//With this function its possible to control a heating pump with the plc
//When the heating pump is switching maualy, then the target power from the ems function is without functionality
//On the max power inputs can be add the power limits. The pump can by step switched by 2 steps
//The percent number from each step is added to the output target power
//< Constants.byTargetOffPowerOnOffDevices Target power from the ems dissable the heating pump after the delay in the surplus mode in Step 4
//When the HP is not step switched, the input target power is set linear to the output target power.
//When the target power from the ems <= 0 and after delay then the heating pump is dissabled in the surplus mode in step 4
//On the emergency power mode and when the soc from the battery <= dissableSOC then the target output power from the heating pump is 0
//Otherwise the heating pump runs in normal mode and the output boutputHB is then always true 
//If in the setups from the heating pump the OffOn Emergency mode is true then the Heating pump is dissabled in the emergency power mode
//When the time function is enabled, then the heating pump run in this time with the % value from max power [1] from the setup when its step switched.
//If there is no step switching and time mode is active, the power input is set linearly to the output. The % value with which the pump should then run over the time can be set at the setups
//This function has also a external look input. If this input is set then the heating pump is dissabled
//This function has also a step to activate the heating pump by a external command. Here the pump switch on with delay and check before the power on the grid

(*---------------------------------------------------------------Limits-------------------------------------------------------------------------------*)

dwBatterySOC := LIMIT(0,dwBatterySOC,100);
	stSetupHP.byManualyTargetPower := LIMIT(0,stSetupHP.byManualyTargetPower,100);
		rBoilerTempHeatingSys := LIMIT(-30,rBoilerTempHeatingSys,120);
			rBoilerTempServiceWater := LIMIT(-30,rBoilerTempServiceWater,120);
				rFlowTemp := LIMIT(-30,rFlowTemp,120);
					rReturnTemp := LIMIT(-30,rReturnTemp,120);
						rFlowTempEnergySource := LIMIT(-30,rFlowTempEnergySource,120); 
							rReturnTempEnergySource := LIMIT(-30,rReturnTempEnergySource,120); 
								stSetupHP.byTimeEnabledTargetPower := LIMIT(0,stSetupHP.byTimeEnabledTargetPower,100);
									stSetupHP.byHourOn := LIMIT(0,stSetupHP.byHourOn,23);
										stSetupHP.byHourOff := LIMIT(0,stSetupHP.byHourOff,23);
											stSetupHP.byMinutesOn := LIMIT(0,stSetupHP.byMinutesOn,59);
												stSetupHP.byMinutesOff := LIMIT(0,stSetupHP.byMinutesOff,59);
													IF IsFinite(F_LREAL(lrCounterThermalEnergy_Water)) THEN lrCounterThermalEnergy_Water := LIMIT(0,lrCounterThermalEnergy_Water,999999999999999); END_IF
														IF IsFinite(F_LREAL(lrCounterThermalEnergy_Heating)) THEN lrCounterThermalEnergy_Heating := LIMIT(0,lrCounterThermalEnergy_Heating,999999999999999); END_IF
															diNumberOfHP := LIMIT(0,diNumberOfHP,Constants_Energy.diMaxNumberOfHeatingPumps);
																tOnDelayExternalOn := LIMIT(T#1M,tOnDelayExternalOn,T#10M);	
																	tOffDelayExternalOn := LIMIT(T#15M,tOffDelayExternalOn,T#2H);
																		tMinOnTime := LIMIT(T#15M,tMinOnTime,T#2H);	

IF IsFinite(F_LREAL(lrTotalCounterEnergy_Consumption)) THEN lrTotalCounterEnergy_Consumption := LIMIT(0,lrTotalCounterEnergy_Consumption,999999999999999); END_IF
	IF IsFinite(F_LREAL(lrTotalCounterEnergy_Production)) THEN lrTotalCounterEnergy_Production := LIMIT(0,lrTotalCounterEnergy_Production,999999999999999); END_IF
		IF IsFinite(F_LREAL(lrCounterEnergyT1_Consumption)) THEN lrCounterEnergyT1_Consumption := LIMIT(0,lrCounterEnergyT1_Consumption,999999999999999); END_IF
			IF IsFinite(F_LREAL(lrCounterEnergyT2_Consumption)) THEN lrCounterEnergyT2_Consumption := LIMIT(0,lrCounterEnergyT2_Consumption,999999999999999); END_IF
				IF IsFinite(F_LREAL(lrCounterEnergyT1_Production)) THEN lrCounterEnergyT1_Production := LIMIT(0,lrCounterEnergyT1_Production,999999999999999); END_IF
					IF IsFinite(F_LREAL(lrCounterEnergyT2_Production)) THEN lrCounterEnergyT2_Production := LIMIT(0,lrCounterEnergyT2_Production,999999999999999); END_IF
						lrElPowerHP := LIMIT(-999999999999999,lrElPowerHP,999999999999999);	
							lrSizeGridConnection := LIMIT(-999999999999999,lrSizeGridConnection,999999999999999);	
								lrGridPower := LIMIT(-999999999999999,lrGridPower,999999999999999);														
														
IF bIsStepSwitched AND stSetupHP.rMaxPower1 <= 0 AND stSetupHP.rMaxPower2 > 0 THEN stSetupHP.rMaxPower1 := stSetupHP.rMaxPower2; END_IF												
												
FOR byLPMaxPower := 1 TO 2 BY 1 DO
	arrTargetPower[byLPMaxPower] := LIMIT(0,arrTargetPower[byLPMaxPower],100);
END_FOR

stSetupHP.rMaxPower1 := LIMIT(0,stSetupHP.rMaxPower1,500);
		stSetupHP.rMaxPower2 := LIMIT(0,stSetupHP.rMaxPower2,500);

//Copy the max input power in the internal array to calculate the steps
arrMaxPower[1] := stSetupHP.rMaxPower1;
	arrMaxPower[2] := stSetupHP.rMaxPower2;
	
IF stSetupHP.byDisableSOC > stSetupHP.byEnableSOC THEN stSetupHP.byEnableSOC := stSetupHP.byDisableSOC + 1; END_IF

stSetupHP.byDisableSOC := LIMIT(0,stSetupHP.byDisableSOC,100);
	stSetupHP.byEnableSOC := LIMIT(1,stSetupHP.byEnableSOC,100);
	
(*---------------------------------------------------------------------------Enable----------------------------------------------------------------------------------*)

stDataHPOut.bEnabled := bEnable;

(*-----------------------------------------------------------------------------Count the steps when the pump is step switched----------------------------------------------------------------------------*)

stDataHPOut.byNumberOfSteps := 0;
	FOR byLPNumberOfSteps := 1 TO 2 BY 1 DO
		IF arrMaxPower[byLPNumberOfSteps] > 0 THEN stDataHPOut.byNumberOfSteps := stDataHPOut.byNumberOfSteps + 1; END_IF
	END_FOR

(*-----------------------------------------------------------------------------Max power for the output----------------------------------------------------------------------------*)	
	
FOR byLPMaxPowerLimit := 1 TO 2 BY 1 DO
	stDataHPOut.arrMaxPower[byLPMaxPowerLimit] := DINT_TO_REAL(REAL_TO_DINT(arrMaxPower[byLPMaxPowerLimit] * 100)) / 100;
END_FOR		
	
(*-----------------------------------------------------------------------------Errors and Warning----------------------------------------------------------------------------*)

FPReset(CLK:= stSetupHP.bReset AND (stDataHPOut.byErrorWarning <> 0), Q=> ); 
	timResetOut(IN:= FPReset.Q AND NOT timResetOut.Q, PT:= T#2S, Q=> stDataHPOut.bSReset, ET=> );
		FPResetIntern(CLK:= bReset, Q=> );	
			IF FPResetIntern.Q THEN stDataHPOut.byErrorWarning := 0; END_IF	 	

IF bWarning AND stDataHPOut.byErrorWarning <> 2 THEN stDataHPOut.byErrorWarning := 1; END_IF
	IF bError THEN stDataHPOut.byErrorWarning := 2; END_IF

//Messages and Error Codes
IF uiState = 3 THEN stDataHPOut.eMessage := E_Message_HP.eExternalOnCommandIsActive;	
ELSIF bExternalLock THEN stDataHPOut.eMessage := E_Message_HP.eExternalLockActive;
ELSIF stDataHPOut.byErrorWarning = 1 AND iWarningCode = 0 THEN stDataHPOut.eMessage := E_Message_HP.eNoConnectionToBackend;
ELSIF stDataHPOut.byErrorWarning = 2 AND iErrorCode = 0 THEN stDataHPOut.eMessage := E_Message_HP.eHPError;
ELSIF stDataHPOut.byErrorWarning = 2 AND iErrorCode = 1 THEN stDataHPOut.eMessage := E_Message_HP.eTooMuchHP;
ELSIF stDataHPOut.byErrorWarning = 2 AND iErrorCode = 2 THEN stDataHPOut.eMessage := E_Message_HP.eWindowsSystemTimeError;
ELSIF stDataHPOut.byErrorWarning = 2 AND iErrorCode = 3 THEN stDataHPOut.eMessage := E_Message_HP.eConnectionError;
ELSE stDataHPOut.eMessage := E_Message_HP.eNoMessage; 
END_IF	
	
(*----------------------------------------------------------------------------Logic------------------------------------------------------------------------------------*)

//Timer for SOC dissabling
timSOCOff(IN:= dwBatterySOC <= stSetupHP.byDisableSOC, PT:= T#30S, Q=> , ET=> );

//Calcualte the % value from each step when the pump is step switched
rSumOfSteps := 0;
	FOR byLPCalcStepPower := 1 TO 2 BY 1 DO
		rSumOfSteps := rSumOfSteps + stDataHPOut.arrMaxPower[byLPCalcStepPower];
			arrPercentValuesSteps[byLPCalcStepPower] := 0;	
	END_FOR
IF stDataHPOut.byNumberOfSteps > 0 AND stDataHPOut.byNumberOfSteps <= 2 AND rSumOfSteps > 0 THEN
	FOR byLPCalcPercentPowerSteps := 1 TO stDataHPOut.byNumberOfSteps BY 1 DO
		arrPercentValuesSteps[byLPCalcPercentPowerSteps] := (stDataHPOut.arrMaxPower[byLPCalcPercentPowerSteps] * 100) / rSumOfSteps;
	END_FOR 
END_IF

arrPercentValuesSteps[1] := DINT_TO_REAL(REAL_TO_DINT(arrPercentValuesSteps[1] * 100)) / 100; 
	arrPercentValuesSteps[2] := DINT_TO_REAL(REAL_TO_DINT(arrPercentValuesSteps[2] * 100)) / 100; 

//Enable the pump about the time function
FPTimeEn(CLK:= stSystemTime.wHour >= stSetupHP.byHourOn AND stSystemTime.wMinute >= stSetupHP.byMinutesOn AND stSetupHP.bTimeEnabled, Q=> );
	FPTimeDis(CLK:= stSystemTime.wHour >= stSetupHP.byHourOff AND stSystemTime.wMinute >= stSetupHP.byMinutesOff AND stSetupHP.bTimeEnabled, Q=> );

IF FPTimeEn.Q THEN bEnableTimeFunction := TRUE; END_IF
	IF FPTimeDis.Q THEN bEnableTimeFunction := FALSE; END_IF	
	
IF NOT stSetupHP.bTimeEnabled THEN bEnableTimeFunction := FALSE; END_IF

//Activate the different operation modes

FPExternalOnCommand(CLK:= bExternalOnCommand, Q=> );

IF bEnable AND NOT bExternalLock AND bEnableTimeFunction AND NOT bIsStepSwitched AND stDataHPOut.byErrorWarning <> 2 THEN uiState := 1; END_IF
IF bEnable AND NOT bExternalLock AND bEnableTimeFunction AND bIsStepSwitched AND stDataHPOut.byErrorWarning <> 2 THEN uiState := 2; END_IF
IF bEnable AND NOT bExternalLock AND NOT bEPOIsActive AND FPExternalOnCommand.Q AND stDataHPOut.byErrorWarning <> 2 THEN uiState := 3; END_IF
IF bEnable AND NOT bExternalLock AND stDataHPOut.byErrorWarning <> 2 AND (arrTargetPower[1] > 0 OR arrTargetPower[2] > 0) THEN uiState := 4; END_IF
IF bEnable AND NOT bExternalLock AND stDataHPOut.byErrorWarning <> 2 AND stSetupHP.bManualyOn THEN uiState := 5; END_IF 

IF NOT bEnable OR stDataHPOut.byErrorWarning = 2 OR bExternalLock THEN uiState := 0; END_IF

//Timer for Min on time in Step 4 in the surplus mode
FPStartMinOnTimer(CLK:= uiState = 4 AND stDataHPOut.rTargetPower > 0 AND bHPIsRunning, Q=> );
	timMinOnInStep4(IN:= FPStartMinOnTimer.Q, PT:= tMinOnTime, Q=> , ET=> );

CASE uiState OF
	
	0: //Init Step and Error
		IF (NOT bEPOIsActive AND bEnable AND NOT bExternalLock AND stDataHPOut.byErrorWarning <> 2) OR 
				(bEPOIsActive AND bEnable AND NOT bExternalLock AND stDataHPOut.byErrorWarning <> 2 AND NOT stSetupHP.bOnEmergPowerOff AND dwBatterySOC >= stSetupHP.byEnableSOC) THEN
					stDataHPOut.bOutput := TRUE;
		END_IF
			IF (bEPOIsActive AND timSOCOff.Q OR NOT bEnable OR bExternalLock OR stDataHPOut.byErrorWarning = 2 OR (bEPOIsActive AND stSetupHP.bOnEmergPowerOff)) THEN
				stDataHPOut.bOutput := FALSE;
					stDataHPOut.rTargetPower := 0;
			END_IF
			
	1: //Enable Heating pump about the time function (linear power)
		//On
		IF (NOT bEPOIsActive AND bEnableTimeFunction AND stSetupHP.byTimeEnabledTargetPower > 0) OR (bEnableTimeFunction AND stSetupHP.byTimeEnabledTargetPower > 0 AND bEPOIsActive AND NOT stSetupHP.bOnEmergPowerOff AND dwBatterySOC >= stSetupHP.byEnableSOC) THEN
			stDataHPOut.bOutput := TRUE; stDataHPOut.rTargetPower := BYTE_TO_REAL(stSetupHP.byTimeEnabledTargetPower);
		END_IF
		//Off		
		IF NOT bEnableTimeFunction OR stSetupHP.byTimeEnabledTargetPower <= 0 OR (bEPOIsActive AND stSetupHP.bOnEmergPowerOff) OR (bEPOIsActive AND (timSOCOff.Q)) THEN 
			stDataHPOut.rTargetPower := 0; 
		END_IF	
			IF stSetupHP.byTimeEnabledTargetPower <= 0 OR (bEPOIsActive AND stSetupHP.bOnEmergPowerOff) OR (bEPOIsActive AND (timSOCOff.Q)) THEN
				stDataHPOut.bOutput := FALSE;
			END_IF	 
		
	2: //Enable Heating pump about the time function (step switched)
		//On
		IF (NOT bEPOIsActive AND bEnableTimeFunction AND arrPercentValuesSteps[1] > 0) OR (bEnableTimeFunction AND arrPercentValuesSteps[1] > 0 AND bEPOIsActive AND NOT stSetupHP.bOnEmergPowerOff AND dwBatterySOC >= stSetupHP.byEnableSOC) THEN
			stDataHPOut.bOutput := TRUE; stDataHPOut.rTargetPower := arrPercentValuesSteps[1];
		END_IF
		//Off
		IF NOT bEnableTimeFunction OR arrPercentValuesSteps[1] <= 0 OR (bEPOIsActive AND stSetupHP.bOnEmergPowerOff) OR (bEPOIsActive AND (timSOCOff.Q)) THEN 
			stDataHPOut.rTargetPower := 0; 
		END_IF	
			IF arrPercentValuesSteps[1] <= 0 OR (bEPOIsActive AND stSetupHP.bOnEmergPowerOff) OR (bEPOIsActive AND (timSOCOff.Q)) THEN
				stDataHPOut.bOutput := FALSE;
			END_IF	 
	 
	3: //Switch on the HP with external on command on max power
		
			CASE iStateIntStep3 OF
				
				0: //Search biggest power from the HP
					//Max Power 1 (1 Step switched or linear/modular)
					IF stSetupHP.rMaxPower1 > 0 AND stSetupHP.rMaxPower2 = 0 THEN
						//Start delay timer when the actual grid power has the capacity for the heating pump max power
						IF (lrGridPower + stSetupHP.rMaxPower1) <= lrSizeGridConnection AND diNumberOfHP > 0 THEN timOnDelayExternalOn.IN := TRUE; ELSE timOnDelayExternalOn.IN := FALSE; END_IF 
					END_IF 
						//Max Power 2 (1 Step switched or linear/modular) 
						IF stSetupHP.rMaxPower2 > 0 AND stSetupHP.rMaxPower1 = 0 THEN 
							//Start delay timer when the actual grid power has the capacity for the heating pump max power
							IF (lrGridPower + stSetupHP.rMaxPower2) <= lrSizeGridConnection AND diNumberOfHP > 0 THEN timOnDelayExternalOn.IN := TRUE; ELSE timOnDelayExternalOn.IN := FALSE; END_IF
						END_IF 
							//Max Power 1 and Max Power 2 (2 Step switched)
							IF stSetupHP.rMaxPower2 > 0 AND stSetupHP.rMaxPower1 > 0 THEN 
								//Start delay timer when the actual grid power has the capacity for the heating pump max power
								IF (lrGridPower + stSetupHP.rMaxPower1 + stSetupHP.rMaxPower2) <= lrSizeGridConnection AND diNumberOfHP > 0 THEN timOnDelayExternalOn.IN := TRUE; ELSE timOnDelayExternalOn.IN := FALSE; END_IF
							END_IF 
								//Next step
								IF timOnDelayExternalOn.Q THEN iStateIntStep3 := 1; timOnDelayExternalOn.IN := FALSE; END_IF
		
				1: //Switch on the Heating pump with max power			
					stDataHPOut.rTargetPower := 100;
						stDataHPOut.bOutput := TRUE;
							stDataHPOut.bExtOnCommandIsActive := TRUE;
								timOffDelayExternalOn.IN := TRUE;
						//Next step
						IF timOffDelayExternalOn.Q THEN iStateIntStep3 := 0; uiState := 0; stDataHPOut.rTargetPower := 0; END_IF 
				
			END_CASE
		
				//Stop this program when the emergency power mode is active
				IF bEPOIsActive THEN uiState := 0; stDataHPOut.rTargetPower := 0; END_IF
					//Stop this programm when we have no power data from the heating pump
					IF stSetupHP.rMaxPower1 >= stSetupHP.rMaxPower2 AND stSetupHP.rMaxPower1 = 0 THEN uiState := 0; stDataHPOut.rTargetPower := 0; END_IF   	
			
	4: //Enable the Heating pump with the target power from the EMS function
		//Power to the heating pump (linear)
		IF NOT bIsStepSwitched AND stDataHPOut.byNumberOfSteps > 0 THEN	
			stDataHPOut.rTargetPower := DINT_TO_REAL(REAL_TO_DINT(arrTargetPower[1] * 100)) / 100;
		END_IF
			//When the min on Time is not passed and the input target power is < 1% then set the output target power to 1%
			IF NOT bIsStepSwitched AND stDataHPOut.byNumberOfSteps > 0 AND arrTargetPower[1] <= 1 AND timMinOnInStep4.Q THEN
				stDataHPOut.rTargetPower := 1;
			END_IF   
		
				//Power to the heating pump (step switched)
				FOR byLPMaxIsReached := 1 TO 2 BY 1 DO
					IF arrTargetPower[byLPMaxIsReached] >= 100 THEN arrMaxIsReached[byLPMaxIsReached] := TRUE; END_IF
						IF arrTargetPower[byLPMaxIsReached] < Constants_Energy.byTargetOffPowerForOnOffDevices THEN arrMaxIsReached[byLPMaxIsReached] := FALSE; END_IF	
				END_FOR
				
				//Off after min on time is passed
				IF NOT timMinOnInStep4.Q AND bIsStepSwitched AND stDataHPOut.byNumberOfSteps > 0 AND NOT arrMaxIsReached[1] AND arrTargetPower[1] < Constants_Energy.byTargetOffPowerForOnOffDevices THEN 
					stDataHPOut.rTargetPower := 0; 
				END_IF
				IF timMinOnInStep4.Q AND bIsStepSwitched AND stDataHPOut.byNumberOfSteps > 0 AND NOT arrMaxIsReached[1] AND arrTargetPower[1] < Constants_Energy.byTargetOffPowerForOnOffDevices THEN 
					stDataHPOut.rTargetPower := arrPercentValuesSteps[1];
				END_IF 
					//Step 1
					IF bIsStepSwitched AND stDataHPOut.byNumberOfSteps > 0 AND arrMaxIsReached[1] AND arrTargetPower[1] >= Constants_Energy.byTargetOffPowerForOnOffDevices THEN 
						stDataHPOut.rTargetPower := arrPercentValuesSteps[1]; 	
					END_IF
						//Step 2
						IF bIsStepSwitched AND stDataHPOut.byNumberOfSteps > 0 AND arrMaxIsReached[1] AND arrMaxIsReached[2] AND arrTargetPower[2] >= Constants_Energy.byTargetOffPowerForOnOffDevices THEN 
							stDataHPOut.rTargetPower := arrPercentValuesSteps[1] + arrPercentValuesSteps[2]; 
						END_IF
						
		IF bIsStepSwitched AND stDataHPOut.rTargetPower > 100 THEN stDataHPOut.rTargetPower := 100; END_IF 
			
		//Switch the outputs
		IF (NOT bEPOIsActive AND stDataHPOut.byNumberOfSteps > 0) OR 
			(bEPOIsActive AND stDataHPOut.byNumberOfSteps > 0 AND NOT stSetupHP.bOnEmergPowerOff AND dwBatterySOC >= stSetupHP.byEnableSOC) THEN
				stDataHPOut.bOutput := TRUE;
		END_IF
			IF (bEPOIsActive AND timSOCOff.Q OR (bEPOIsActive AND stSetupHP.bOnEmergPowerOff)) OR 
				stDataHPOut.byNumberOfSteps <= 0 THEN
					stDataHPOut.bOutput := FALSE;
			END_IF 	
		
		IF NOT stDataHPOut.bOutput THEN stDataHPOut.rTargetPower := 0; END_IF 

	5: //Switch manually
		stDataHPOut.rTargetPower := BYTE_TO_REAL(stSetupHP.byManualyTargetPower);
		
		IF stSetupHP.bManualyOn AND stDataHPOut.rTargetPower > 0 THEN stDataHPOut.bOutput := TRUE; END_IF
			IF NOT stSetupHP.bManualyOn OR stDataHPOut.rTargetPower <= 0 THEN stDataHPOut.bOutput := FALSE; END_IF 

		IF NOT stDataHPOut.bOutput THEN stDataHPOut.rTargetPower := 0; END_IF 		

END_CASE

//Timer for external command
IF uiState <> 3 THEN timOnDelayExternalOn.IN := FALSE; timOffDelayExternalOn.IN := FALSE; iStateIntStep3 := 0; stDataHPOut.bExtOnCommandIsActive := FALSE; END_IF

timOnDelayExternalOn(IN:= , PT:= tOnDelayExternalOn * diNumberOfHP, Q=> , ET=> );
	timOffDelayExternalOn(IN:= , PT:= tOffDelayExternalOn, Q=> , ET=> );
	
(*------------------------------------------------------------------Power Data----------------------------------------------------------------------------------------------*)

IF bEnable THEN
	stDataHPOut.lrElPower:= LINT_TO_LREAL(LREAL_TO_LINT((lrElPowerHP / 1000) * 100)) / 100;
		IF IsFinite(F_LREAL(lrCounterEnergyT1_Consumption)) THEN stDataHPOut.lrCounterEnergyT1_Consumption := LINT_TO_LREAL(LREAL_TO_LINT((lrCounterEnergyT1_Consumption / 1000) * 100)) / 100; END_IF
			IF IsFinite(F_LREAL(lrCounterEnergyT2_Consumption)) THEN stDataHPOut.lrCounterEnergyT2_Consumption := LINT_TO_LREAL(LREAL_TO_LINT((lrCounterEnergyT2_Consumption / 1000) * 100)) / 100; END_IF
				IF IsFinite(F_LREAL(lrCounterEnergyT1_Production)) THEN stDataHPOut.lrCounterEnergyT1_Production := LINT_TO_LREAL(LREAL_TO_LINT((lrCounterEnergyT1_Production / 1000) * 100)) / 100; END_IF
					IF IsFinite(F_LREAL(lrCounterEnergyT2_Production)) THEN stDataHPOut.lrCounterEnergyT2_Production := LINT_TO_LREAL(LREAL_TO_LINT((lrCounterEnergyT2_Production / 1000) * 100)) / 100; END_IF
						IF IsFinite(F_LREAL(lrTotalCounterEnergy_Consumption)) THEN stDataHPOut.lrTotalCounterEnergy_Consumption := LINT_TO_LREAL(LREAL_TO_LINT((lrTotalCounterEnergy_Consumption / 1000) * 100)) / 100; END_IF
							IF IsFinite(F_LREAL(lrTotalCounterEnergy_Production)) THEN stDataHPOut.lrTotalCounterEnergy_Production := LINT_TO_LREAL(LREAL_TO_LINT((lrTotalCounterEnergy_Production / 1000) * 100)) / 100; END_IF 
				
		IF stDataHPOut.lrElPower < 0 THEN
				stDataHPOut.lrElPowerProduction := (stDataHPOut.lrElPower * - 1);
				stDataHPOut.lrElPowerConsumption := 0;
		ELSIF stDataHPOut.lrElPower > 0 THEN
				stDataHPOut.lrElPowerProduction := 0;
				stDataHPOut.lrElPowerConsumption := stDataHPOut.lrElPower;
		ELSIF stDataHPOut.lrElPower = 0 THEN
				stDataHPOut.lrElPowerProduction := 0;
				stDataHPOut.lrElPowerConsumption := 0;
		END_IF
		
ELSE
	stDataHPOut.lrElPower := 0;
		stDataHPOut.lrCounterEnergyT1_Consumption := 0;
			stDataHPOut.lrCounterEnergyT2_Consumption := 0;
				stDataHPOut.lrCounterEnergyT1_Production := 0;
					stDataHPOut.lrCounterEnergyT2_Production := 0;
						stDataHPOut.lrElPowerProduction := 0;
							stDataHPOut.lrElPowerConsumption := 0;	
								stDataHPOut.lrTotalCounterEnergy_Consumption := 0;
									stDataHPOut.lrTotalCounterEnergy_Production := 0;
END_IF

(*---------------------------------------------------------------------------Outputs--------------------------------------------------------------------------------------*)

stDataHPOut.byPriority := stSetupHP.byPriority;
	stDataHPOut.bIsStepSwitched := bIsStepSwitched;
		stDataHPOut.bSOnEmergPowerOff := stSetupHP.bOnEmergPowerOff;
			stDataHPOut.bSManualyOn := stSetupHP.bManualyOn;
				stDataHPOut.bySManualyTargetPower := stSetupHP.byManualyTargetPower;
					stDataHPOut.bSTimeEnabled := stSetupHP.bTimeEnabled;
						stDataHPOut.bySTimeEnabledTargetPower := stSetupHP.byTimeEnabledTargetPower;
				
IF bEnable THEN
	stDataHPOut.rBoilerTempServiceWater := DINT_TO_REAL(REAL_TO_DINT(rBoilerTempServiceWater * 100)) / 100;
		stDataHPOut.rBoilerTempHeatingSys := DINT_TO_REAL(REAL_TO_DINT(rBoilerTempHeatingSys * 100)) / 100;
			stDataHPOut.rReturnTemp := DINT_TO_REAL(REAL_TO_DINT(rReturnTemp * 100)) / 100;
				stDataHPOut.rReturnTempEnergySource := DINT_TO_REAL(REAL_TO_DINT(rReturnTempEnergySource * 100)) / 100;
					stDataHPOut.rFlowTemp := DINT_TO_REAL(REAL_TO_DINT(rFlowTemp * 100)) / 100;
						stDataHPOut.rFlowTempEnergySource := DINT_TO_REAL(REAL_TO_DINT(rFlowTempEnergySource * 100)) / 100;
							IF IsFinite(F_LREAL(lrCounterThermalEnergy_Heating)) THEN stDataHPOut.lrCounterThermalHeatingSys := LINT_TO_LREAL(LREAL_TO_LINT((lrCounterThermalEnergy_Heating / 1000) * 100)) / 100; END_IF
								IF IsFinite(F_LREAL(lrCounterThermalEnergy_Water)) THEN stDataHPOut.lrCounterThermalServiceWater := LINT_TO_LREAL(LREAL_TO_LINT((lrCounterThermalEnergy_Water / 1000) * 100)) / 100; END_IF	
ELSE	
	stDataHPOut.rBoilerTempServiceWater := 0;
		stDataHPOut.rBoilerTempHeatingSys := 0;
			stDataHPOut.rReturnTemp := 0;
				stDataHPOut.rReturnTempEnergySource := 0;
					stDataHPOut.rFlowTemp := 0;
						stDataHPOut.rFlowTempEnergySource := 0;
							stDataHPOut.lrCounterThermalHeatingSys := 0;
								stDataHPOut.lrCounterThermalServiceWater := 0;		
END_IF

timDelayOutputs(IN:= bWriteWithDelay AND bEnable AND NOT timDelayOutputs.Q, PT:= tTimDelayOutput, Q=> , ET=> );
	FPEnable(CLK:= bEnable, Q=> );
		FNEnable(CLK:= bEnable, Q=> );
		
//Write with Delay or without
IF (bWriteWithDelay AND (timDelayOutputs.Q OR FPEnable.Q OR FNEnable.Q)) OR NOT bWriteWithDelay THEN
	stDataHPOutDelay := stDataHPOut;
END_IF

END_FUNCTION_BLOCK

// ---- Energy/FBs Internal/House/FB_HouseConsumption.TcPOU
{attribute 'hide_all_locals'}
{attribute 'conditionalshow'}
FUNCTION_BLOCK FB_HouseConsumption
VAR_INPUT
	{attribute 'hide'}
	bEnable								: BOOL;							//Enable or disable this function
	{attribute 'hide'}
	bError								: BOOL;							//Error from the house consumption
	{attribute 'hide'}
	bWarning							: BOOL;							//Warning from the house consumption
	{attribute 'hide'}
	bWriteWithDelay						: BOOL;							//Write with Delay the Data to the output (Not al Output Data is writen with Delay)
	{attribute 'hide'}
	iErrorCode							: INT;							//Error Code from external House Consumption
	{attribute 'hide'}
	iWarningCode						: INT;							//Warning Code from external House Consumption
	{attribute 'hide'}
	lrTotalCounterEnergy_Consumption	: LREAL;						//Total Counter for Energy consumption with unit Wh
	{attribute 'hide'}
	lrTotalCounterEnergy_Production		: LREAL;						//Total Counter for Energy production with unit Wh
	{attribute 'hide'}
	lrCounterEnergyT1_Consumption		: LREAL;						//Total counter for energy Tariff 1 consumption with unit Wh
	{attribute 'hide'}
	lrCounterEnergyT2_Consumption		: LREAL;						//Total counter for energy Tariff 2 consumption with unit Wh
	{attribute 'hide'}
	lrCounterEnergyT1_Production		: LREAL;						//Total counter for energy Tariff 1 production with unit Wh
	{attribute 'hide'}
	lrCounterEnergyT2_Production		: LREAL;						//Total counter for energy Tariff 2 production with unit Wh
	{attribute 'hide'}
	lrPowerHouseConsumption				: LREAL;						//Input Value from the power of the House with unit W
	{attribute 'hide'}
	tTimDelayOutput						: TIME := T#5S;					//Delay Time to write some Data to the Output
END_VAR
VAR_OUTPUT
	{attribute 'hide'}
	stDataHouseCOut						: ST_HouseConsumption_Output;	//House consumption output data
	{attribute 'hide'}
	stDataHouseCOutDelay				: ST_HouseConsumption_Output;	//House consumption output data with delay
END_VAR
VAR	
	FPEnable							: R_TRIG;						//Internal positive Edge
	FNEnable							: F_TRIG;						//Internal negative Edge
	timDelayOutputs						: TON;							//Timer to send Data with Delay to the outputs
END_VAR

//Creator : Kai Ebensperger
//Company : Lynus AG
//Date : 29.05.2021
//Version : 1.0.0.0

//With this function its possible to handle the most important values from a hous consumption

(*---------------------------------------------------------------Check the limits of the inputs-------------------------------------------------------------------------------*)

IF IsFinite(F_LREAL(lrTotalCounterEnergy_Consumption)) THEN lrTotalCounterEnergy_Consumption := LIMIT(0,lrTotalCounterEnergy_Consumption,999999999999999); END_IF
	IF IsFinite(F_LREAL(lrTotalCounterEnergy_Production)) THEN lrTotalCounterEnergy_Production := LIMIT(0,lrTotalCounterEnergy_Production,999999999999999); END_IF
		IF IsFinite(F_LREAL(lrCounterEnergyT1_Consumption)) THEN lrCounterEnergyT1_Consumption := LIMIT(0,lrCounterEnergyT1_Consumption,999999999999999); END_IF
			IF IsFinite(F_LREAL(lrCounterEnergyT2_Consumption)) THEN lrCounterEnergyT2_Consumption := LIMIT(0,lrCounterEnergyT2_Consumption,999999999999999); END_IF
				IF IsFinite(F_LREAL(lrCounterEnergyT1_Production)) THEN lrCounterEnergyT1_Production := LIMIT(0,lrCounterEnergyT1_Production,999999999999999); END_IF
					IF IsFinite(F_LREAL(lrCounterEnergyT2_Production)) THEN lrCounterEnergyT2_Production := LIMIT(0,lrCounterEnergyT2_Production,999999999999999); END_IF
						lrPowerHouseConsumption := LIMIT(-999999999999999,lrPowerHouseConsumption,999999999999999);

(*---------------------------------------------------------------Enable-------------------------------------------------------------------------------*)
stDataHouseCOut.bEnabled := bEnable;

(*---------------------------------------------------------------Power data-------------------------------------------------------------------------------*)

timDelayOutputs(IN:= bWriteWithDelay AND bEnable AND NOT timDelayOutputs.Q, PT:= tTimDelayOutput, Q=> , ET=> );
	FPEnable(CLK:= bEnable, Q=> );
		FNEnable(CLK:= bEnable, Q=> );

IF bEnable THEN
	stDataHouseCOut.lrPower:= LINT_TO_LREAL(LREAL_TO_LINT((lrPowerHouseConsumption / 1000) * 100)) / 100;
		IF IsFinite(F_LREAL(lrCounterEnergyT1_Consumption)) THEN stDataHouseCOut.lrCounterEnergyT1_Consumption := LINT_TO_LREAL(LREAL_TO_LINT((lrCounterEnergyT1_Consumption / 1000) * 100)) / 100; END_IF
			IF IsFinite(F_LREAL(lrCounterEnergyT2_Consumption)) THEN stDataHouseCOut.lrCounterEnergyT2_Consumption := LINT_TO_LREAL(LREAL_TO_LINT((lrCounterEnergyT2_Consumption / 1000) * 100)) / 100; END_IF
				IF IsFinite(F_LREAL(lrCounterEnergyT1_Production)) THEN stDataHouseCOut.lrCounterEnergyT1_Production := LINT_TO_LREAL(LREAL_TO_LINT((lrCounterEnergyT1_Production / 1000) * 100)) / 100; END_IF
					IF IsFinite(F_LREAL(lrCounterEnergyT2_Production)) THEN stDataHouseCOut.lrCounterEnergyT2_Production := LINT_TO_LREAL(LREAL_TO_LINT((lrCounterEnergyT2_Production / 1000) * 100)) / 100; END_IF
						IF IsFinite(F_LREAL(lrTotalCounterEnergy_Consumption)) THEN stDataHouseCOut.lrTotalCounterEnergy_Consumption := LINT_TO_LREAL(LREAL_TO_LINT((lrTotalCounterEnergy_Consumption / 1000) * 100)) / 100; END_IF
							IF IsFinite(F_LREAL(lrTotalCounterEnergy_Production)) THEN stDataHouseCOut.lrTotalCounterEnergy_Production := LINT_TO_LREAL(LREAL_TO_LINT((lrTotalCounterEnergy_Production / 1000) * 100)) / 100; END_IF 	 
				
		IF stDataHouseCOut.lrPower < 0 THEN
				stDataHouseCOut.lrPowerProduction := (stDataHouseCOut.lrPower * - 1);
				stDataHouseCOut.lrPowerConsumption := 0;
		ELSIF stDataHouseCOut.lrPower > 0 THEN
				stDataHouseCOut.lrPowerProduction := 0;
				stDataHouseCOut.lrPowerConsumption := stDataHouseCOut.lrPower;
		ELSIF stDataHouseCOut.lrPower = 0 THEN
				stDataHouseCOut.lrPowerProduction := 0;
				stDataHouseCOut.lrPowerConsumption := 0;
		END_IF															
ELSE																			
	stDataHouseCOut.lrPower := 0;
		stDataHouseCOut.lrCounterEnergyT1_Consumption := 0;
			stDataHouseCOut.lrCounterEnergyT2_Consumption := 0;
				stDataHouseCOut.lrCounterEnergyT1_Production := 0;
					stDataHouseCOut.lrCounterEnergyT2_Production := 0;
						stDataHouseCOut.lrPowerProduction := 0;
							stDataHouseCOut.lrPowerConsumption := 0;
								stDataHouseCOut.lrTotalCounterEnergy_Consumption := 0;
									stDataHouseCOut.lrTotalCounterEnergy_Production := 0;
END_IF	

(*---------------------------------------------------------------Error and Warning-------------------------------------------------------------------------------*)

stDataHouseCOut.byErrorWarning := 0;
	IF bWarning THEN stDataHouseCOut.byErrorWarning := 1; END_IF
	IF bError THEN stDataHouseCOut.byErrorWarning := 2; END_IF

//Messages and Error Codes
IF stDataHouseCOut.byErrorWarning = 1 AND iWarningCode = 0 THEN stDataHouseCOut.eMessage := E_Message_HouseC.eNoConnectionToBackend;
ELSIF stDataHouseCOut.byErrorWarning = 2 AND iErrorCode = 0 THEN stDataHouseCOut.eMessage := E_Message_HouseC.eErrorHouseC;
ELSIF stDataHouseCOut.byErrorWarning = 2 AND iErrorCode = 1 THEN stDataHouseCOut.eMessage := E_Message_HouseC.eTooMuchHouseC;
ELSE stDataHouseCOut.eMessage := E_Message_HouseC.eNoMessage; 
END_IF

(*---------------------------------------------------------------Outputs-------------------------------------------------------------------------------*)

//Write with Delay or without
IF (bWriteWithDelay AND (timDelayOutputs.Q OR FPEnable.Q OR FNEnable.Q)) OR NOT bWriteWithDelay THEN
	stDataHouseCOutDelay := stDataHouseCOut; 
END_IF

END_FUNCTION_BLOCK

// ---- Energy/FBs Internal/Other Big Consumer/FB_BigConsumer.TcPOU
{attribute 'hide_all_locals'}
{attribute 'conditionalshow'}
FUNCTION_BLOCK FB_BigConsumer
VAR_INPUT
	{attribute 'hide'}
	bEnable								: BOOL;									//Enable or dissable this function
	{attribute 'hide'}
	bError								: BOOL;									//Error from the big consumer
	{attribute 'hide'}
	bWarning							: BOOL;									//Warning from the big consumer
	{attribute 'hide'}
	bEPOIsActive						: BOOL;									//Emergency power operation is active
	{attribute 'hide'}
	bExternalLock						: BOOL;									//External lock (All functions are locked)
	{attribute 'hide'}
	bWriteWithDelay						: BOOL;									//Write with Delay the Data to the output (Not al Output Data is writen with Delay)
	{attribute 'hide'}
	iErrorCode							: INT;									//Error Code from external OBC
	{attribute 'hide'}
	iWarningCode						: INT;									//Warning Code from external OBC
	{attribute 'hide'}
	dwBatterySOC						: DWORD;								//Actual Battery SOC in %
	{attribute 'hide'}
	lrTotalCounterEnergy_Consumption	: LREAL;								//Total Counter for Energy consumption with unit Wh
	{attribute 'hide'}
	lrTotalCounterEnergy_Production		: LREAL;								//Total Counter for Energy production with unit Wh
	{attribute 'hide'}
	lrCounterEnergyT1_Consumption		: LREAL;								//Total counter for energy Tariff 1 consumption with unit Wh
	{attribute 'hide'}
	lrCounterEnergyT2_Consumption		: LREAL;								//Total counter for energy Tariff 2 consumption with unit Wh
	{attribute 'hide'}
	lrCounterEnergyT1_Production		: LREAL;								//Total counter for energy Tariff 1 production with unit Wh
	{attribute 'hide'}
	lrCounterEnergyT2_Production		: LREAL;								//Total counter for energy Tariff 2 production with unit Wh
	{attribute 'hide'}
	lrPowerOBC							: LREAL;								//Input Value from the power of the big consumer with unit W
	{attribute 'hide'}
	rTargetPower						: REAL;									//Target power from 0% to +100%
	{attribute 'hide'}
	tTimDelayOutput						: TIME := T#5S;							//Delay Time to write some Data to the Output	
	{attribute 'hide'}
	stSetupOBC							: ST_Setup_OBC;							//Setup other big consumer
END_VAR
VAR_OUTPUT
	{attribute 'hide'}
	stDataOBCOut						: ST_OBC_Output;						//Other big consumer output data
	{attribute 'hide'}
	stDataOBCOutDelay					: ST_OBC_Output;						//Other big consumer output data with delay
END_VAR
VAR
	FPEnable							: R_TRIG;								//Internal positive Edge
	FNEnable							: F_TRIG;								//Internal negative Edge
	FNManualy							: F_TRIG;								//Internal negative edge
	timDelayOutputs						: TON;									//Timer to send Data with Delay to the outputs
	timSOCOff							: TON;									//Timer to dissable the Device when the SOC from the Battery is under the Setpoint
	timError							: TOF;									//Timer to set the error
END_VAR

//Creator : Kai Ebensperger
//Company : Lynus AG
//Date : 29.05.2021
//Version : 1.0.0.0

//With this function its possible to control a other big consumer with the plc
//When the big consumer is switching maualy, then the target power from the ems function is without functionality
//The output from the big consumer will be set when the target power from the ems is >= 100%
//When the target power is < Constants.byTargetOffPowerOnOffDevices then the output for On/Off will be reset
//When the big consumer is controllable then the target power is set linear to the output
//When the big consumer is controlled by the target power mode, then the soc from the battery must have a value between the On soc and Off soc fromt he setups and the On soc must be reached on time to enable the big consumer. 
//Optional this function has a external lock possibility. If this lock is active, then the big consumer is off and without functionality.  
//When the system is in emergency power mode, then its possible to switch off this big consumer automatically.

(*---------------------------------------------------------------Limits-------------------------------------------------------------------------------*)

stSetupOBC.rMaxPower := LIMIT(0,stSetupOBC.rMaxPower,500);
	rTargetPower := LIMIT(0,rTargetPower,100);
		dwBatterySOC := LIMIT(0,dwBatterySOC,100);
			stSetupOBC.byManualyTargetPower := LIMIT(0,stSetupOBC.byManualyTargetPower,100);

IF IsFinite(F_LREAL(lrTotalCounterEnergy_Consumption)) THEN lrTotalCounterEnergy_Consumption := LIMIT(0,lrTotalCounterEnergy_Consumption,999999999999999); END_IF
	IF IsFinite(F_LREAL(lrTotalCounterEnergy_Production)) THEN lrTotalCounterEnergy_Production := LIMIT(0,lrTotalCounterEnergy_Production,999999999999999); END_IF
		IF IsFinite(F_LREAL(lrCounterEnergyT1_Consumption)) THEN lrCounterEnergyT1_Consumption := LIMIT(0,lrCounterEnergyT1_Consumption,999999999999999); END_IF
			IF IsFinite(F_LREAL(lrCounterEnergyT2_Consumption)) THEN lrCounterEnergyT2_Consumption := LIMIT(0,lrCounterEnergyT2_Consumption,999999999999999); END_IF
				IF IsFinite(F_LREAL(lrCounterEnergyT1_Production)) THEN lrCounterEnergyT1_Production := LIMIT(0,lrCounterEnergyT1_Production,999999999999999); END_IF
					IF IsFinite(F_LREAL(lrCounterEnergyT2_Production)) THEN lrCounterEnergyT2_Production := LIMIT(0,lrCounterEnergyT2_Production,999999999999999); END_IF
						lrPowerOBC := LIMIT(-999999999999999,lrPowerOBC,999999999999999);
				
IF stSetupOBC.byDisableSOC > stSetupOBC.byEnableSOC THEN stSetupOBC.byEnableSOC := stSetupOBC.byDisableSOC + 1; END_IF

stSetupOBC.byDisableSOC := LIMIT(0,stSetupOBC.byDisableSOC,100);
	stSetupOBC.byEnableSOC := LIMIT(1,stSetupOBC.byEnableSOC,100);

(*---------------------------------------------------------------Enable-------------------------------------------------------------------------------*)

stDataOBCOut.bEnabled := bEnable;

(*---------------------------------------------------------------Error and Waring-------------------------------------------------------------------------------*)

timError(IN:= bError, PT:= T#5S, Q=> , ET=> );

stDataOBCOut.byErrorWarning := 0;
	IF bWarning THEN stDataOBCOut.byErrorWarning := 1; END_IF 
	IF timError.Q THEN stDataOBCOut.byErrorWarning := 2; END_IF

//Messages and Error Codes
IF bExternalLock THEN stDataOBCOut.eMessage := E_Message_OBC.eExternalLockActive;
ELSIF stDataOBCOut.byErrorWarning = 1 AND iWarningCode = 0 THEN stDataOBCOut.eMessage := E_Message_OBC.eNoConnectionToBackend;
ELSIF stDataOBCOut.byErrorWarning = 2 AND iErrorCode = 0 THEN stDataOBCOut.eMessage := E_Message_OBC.eErrorOBC;
ELSIF stDataOBCOut.byErrorWarning = 2 AND iErrorCode = 1 THEN stDataOBCOut.eMessage := E_Message_OBC.eTooMuchOBC;
ELSE stDataOBCOut.eMessage := E_Message_OBC.eNoMessage; 
END_IF

(*---------------------------------------------------------------Logic-------------------------------------------------------------------------------*)

//Timer for SOC dissabling
timSOCOff(IN:= dwBatterySOC <= stSetupOBC.byDisableSOC, PT:= T#30S, Q=> , ET=> );

//Target power
stDataOBCOut.rTargetPower := DINT_TO_REAL(REAL_TO_DINT(rTargetPower * 100)) / 100;
IF stSetupOBC.bManualyOn THEN stDataOBCOut.rTargetPower := BYTE_TO_REAL(stSetupOBC.byManualyTargetPower); END_IF

 //Switch off
FNManualy(CLK:= stSetupOBC.bManualyOn, Q=> ); 
 
IF NOT bEnable OR bExternalLock OR stDataOBCOut.byErrorWarning = 2 OR stDataOBCOut.rTargetPower <= 0 OR timSOCOff.Q OR (bEPOIsActive AND stSetupOBC.bOnEmergPowerOff) OR FNManualy.Q THEN
	stDataOBCOut.bOutput := FALSE;
END_IF

//Switch On
IF (bEnable AND NOT bExternalLock AND stDataOBCOut.byErrorWarning <> 2 AND NOT bEPOIsActive AND rTargetPower > 0 AND dwBatterySOC >= stSetupOBC.byEnableSOC) OR 
	(bEnable AND NOT bExternalLock AND stDataOBCOut.byErrorWarning <> 2 AND bEPOIsActive AND NOT stSetupOBC.bOnEmergPowerOff AND rTargetPower > 0 AND dwBatterySOC >= stSetupOBC.byEnableSOC) OR
		(bEnable AND NOT bExternalLock AND stDataOBCOut.byErrorWarning <> 2 AND stSetupOBC.bManualyOn) THEN				
			stDataOBCOut.bOutput := TRUE; 
 END_IF

 //Use this Output to switch Charging station on and off without possibility to send a target power value (Not controllable)
IF stDataOBCOut.rTargetPower >= 100 AND stDataOBCOut.bOutput THEN stDataOBCOut.bOutputOnOff := TRUE; END_IF  
IF stDataOBCOut.rTargetPower < Constants_Energy.byTargetOffPowerForOnOffDevices OR NOT stDataOBCOut.bOutput THEN stDataOBCOut.bOutputOnOff := FALSE; END_IF  

IF NOT stDataOBCOut.bOutput THEN stDataOBCOut.rTargetPower := 0; END_IF 
 
(*---------------------------------------------------------------Power data-------------------------------------------------------------------------------*)

IF bEnable THEN
	stDataOBCOut.lrPower := LINT_TO_LREAL(LREAL_TO_LINT((lrPowerOBC / 1000) * 100)) / 100;
		IF IsFinite(F_LREAL(lrCounterEnergyT1_Consumption)) THEN stDataOBCOut.lrCounterEnergyT1_Consumption := LINT_TO_LREAL(LREAL_TO_LINT((lrCounterEnergyT1_Consumption / 1000) * 100)) / 100; END_IF
			IF IsFinite(F_LREAL(lrCounterEnergyT2_Consumption)) THEN stDataOBCOut.lrCounterEnergyT2_Consumption := LINT_TO_LREAL(LREAL_TO_LINT((lrCounterEnergyT2_Consumption / 1000) * 100)) / 100; END_IF
				IF IsFinite(F_LREAL(lrCounterEnergyT1_Production)) THEN stDataOBCOut.lrCounterEnergyT1_Production := LINT_TO_LREAL(LREAL_TO_LINT((lrCounterEnergyT1_Production / 1000) * 100)) / 100; END_IF
					IF IsFinite(F_LREAL(lrCounterEnergyT2_Production)) THEN stDataOBCOut.lrCounterEnergyT2_Production := LINT_TO_LREAL(LREAL_TO_LINT((lrCounterEnergyT2_Production / 1000) * 100)) / 100; END_IF
						IF IsFinite(F_LREAL(lrTotalCounterEnergy_Consumption)) THEN stDataOBCOut.lrTotalCounterEnergy_Consumption := LINT_TO_LREAL(LREAL_TO_LINT((lrTotalCounterEnergy_Consumption / 1000) * 100)) / 100; END_IF
							IF IsFinite(F_LREAL(lrTotalCounterEnergy_Production)) THEN stDataOBCOut.lrTotalCounterEnergy_Production := LINT_TO_LREAL(LREAL_TO_LINT((lrTotalCounterEnergy_Production / 1000) * 100)) / 100; END_IF   
				
		IF stDataOBCOut.lrPower < 0 THEN
				stDataOBCOut.lrPowerProduction := (stDataOBCOut.lrPower * - 1);
				stDataOBCOut.lrPowerConsumption := 0;
		ELSIF stDataOBCOut.lrPower > 0 THEN
				stDataOBCOut.lrPowerProduction := 0;
				stDataOBCOut.lrPowerConsumption := stDataOBCOut.lrPower;
		ELSIF stDataOBCOut.lrPower = 0 THEN
				stDataOBCOut.lrPowerProduction := 0;
				stDataOBCOut.lrPowerConsumption := 0;
		END_IF
		
ELSE
	stDataOBCOut.lrPower := 0;
		stDataOBCOut.lrCounterEnergyT1_Consumption := 0;
			stDataOBCOut.lrCounterEnergyT2_Consumption := 0;
				stDataOBCOut.lrCounterEnergyT1_Production := 0;
					stDataOBCOut.lrCounterEnergyT2_Production := 0;
						stDataOBCOut.lrPowerProduction := 0;
							stDataOBCOut.lrPowerConsumption := 0;	
								stDataOBCOut.lrTotalCounterEnergy_Consumption := 0;
									stDataOBCOut.lrTotalCounterEnergy_Production := 0;
END_IF

(*---------------------------------------------------------------Outputs-------------------------------------------------------------------------------*)

stDataOBCOut.byPriority := stSetupOBC.byPriority;
	stDataOBCOut.rMaxPower := DINT_TO_REAL(REAL_TO_DINT(stSetupOBC.rMaxPower * 100)) / 100;
		stDataOBCOut.bSOnEmergPowerOff := stSetupOBC.bOnEmergPowerOff;
			stDataOBCOut.bSManualyOn := stSetupOBC.bManualyOn;
				stDataOBCOut.bySManualyTargetPower := stSetupOBC.byManualyTargetPower;
				
timDelayOutputs(IN:= bWriteWithDelay AND bEnable AND NOT timDelayOutputs.Q, PT:= tTimDelayOutput, Q=> , ET=> );
	FPEnable(CLK:= bEnable, Q=> );
		FNEnable(CLK:= bEnable, Q=> );
		
//Write with Delay or without
IF (bWriteWithDelay AND (timDelayOutputs.Q OR FPEnable.Q OR FNEnable.Q)) OR NOT bWriteWithDelay THEN
	stDataOBCOutDelay := stDataOBCOut;
END_IF

END_FUNCTION_BLOCK

// ---- Energy/FBs Internal/PV/FB_PV_Production.TcPOU
{attribute 'hide_all_locals'}
{attribute 'conditionalshow'}
FUNCTION_BLOCK FB_PV_Production
VAR_INPUT
	{attribute 'hide'}
	bEnable								: BOOL;						//Enable or dissable the function
	{attribute 'hide'}
	bError								: BOOL;						//Error Pv system
	{attribute 'hide'}
	bWarning							: BOOL;						//Warning Pv system
	{attribute 'hide'}
	bWriteWithDelay						: BOOL;						//Write with Delay the Data to the output (Not al Output Data is writen with Delay)
	{attribute 'hide'}
	iErrorCode							: INT;						//Error Code from external PV
	{attribute 'hide'}
	iWarningCode						: INT;						//Warning Code from external PV
	{attribute 'hide'}
	lrTotalCounterEnergy_Consumption	: LREAL;					//Total Counter for Energy consumption with unit Wh
	{attribute 'hide'}
	lrTotalCounterEnergy_Production		: LREAL;					//Total Counter for Energy production with unit Wh
	{attribute 'hide'}
	lrCounterEnergyT1_Consumption		: LREAL;					//Total counter for energy Tariff 1 consumption with unit Wh
	{attribute 'hide'}
	lrCounterEnergyT2_Consumption		: LREAL;					//Total counter for energy Tariff 2 consumption with unit Wh
	{attribute 'hide'}
	lrCounterEnergyT1_Production		: LREAL;					//Total counter for energy Tariff 1 production with unit Wh
	{attribute 'hide'}
	lrCounterEnergyT2_Production		: LREAL;					//Total counter for energy Tariff 2 production with unit Wh
	{attribute 'hide'}
	lrPvPower							: LREAL;					//Input Value from the power of the Pv system with unit W
	{attribute 'hide'}
	tTimDelayOutput						: TIME := T#5S;				//Delay Time to write some Data to the Output
END_VAR
VAR_OUTPUT
	{attribute 'hide'}
	stDataPvOut							: ST_PV_Output;				//Pv system output data
	{attribute 'hide'}
	stDataPvOutDelay					: ST_PV_Output;				//Pv system output data with delay
END_VAR
VAR
	FPEnable							: R_TRIG;					//Internal positive Edge
	FNEnable							: F_TRIG;					//Internal negative Edge
	timDelayOutputs						: TON;						//Timer to send Data with Delay to the outputs
END_VAR

//Creator : Kai Ebensperger
//Company : Lynus AG
//Date : 29.05.2021
//Version : 1.0.0.0

//With this function its possible to handel the most popular values from a pv system

(*---------------------------------------------------------------Check the limits of the inputs-------------------------------------------------------------------------------*)

IF IsFinite(F_LREAL(lrTotalCounterEnergy_Consumption)) THEN lrTotalCounterEnergy_Consumption := LIMIT(0,lrTotalCounterEnergy_Consumption,999999999999999); END_IF
	IF IsFinite(F_LREAL(lrTotalCounterEnergy_Production)) THEN lrTotalCounterEnergy_Production := LIMIT(0,lrTotalCounterEnergy_Production,999999999999999); END_IF
		IF IsFinite(F_LREAL(lrCounterEnergyT1_Consumption)) THEN lrCounterEnergyT1_Consumption := LIMIT(0,lrCounterEnergyT1_Consumption,999999999999999); END_IF
			IF IsFinite(F_LREAL(lrCounterEnergyT2_Consumption)) THEN lrCounterEnergyT2_Consumption := LIMIT(0,lrCounterEnergyT2_Consumption,999999999999999); END_IF
				IF IsFinite(F_LREAL(lrCounterEnergyT1_Production)) THEN lrCounterEnergyT1_Production := LIMIT(0,lrCounterEnergyT1_Production,999999999999999); END_IF
					IF IsFinite(F_LREAL(lrCounterEnergyT2_Production)) THEN lrCounterEnergyT2_Production := LIMIT(0,lrCounterEnergyT2_Production,999999999999999); END_IF
						lrPvPower := LIMIT(-999999999999999,lrPvPower,999999999999999);

(*---------------------------------------------------------------Enable-------------------------------------------------------------------------------*)
stDataPvOut.bEnabled := bEnable;

(*---------------------------------------------------------------Power data-------------------------------------------------------------------------------*)

timDelayOutputs(IN:= bWriteWithDelay AND bEnable AND NOT timDelayOutputs.Q, PT:= tTimDelayOutput, Q=> , ET=> );
	FPEnable(CLK:= bEnable, Q=> );
		FNEnable(CLK:= bEnable, Q=> );

IF bEnable THEN
	stDataPvOut.lrPower := LINT_TO_LREAL(LREAL_TO_LINT((lrPvPower / 1000) * 100)) / 100;
		IF IsFinite(F_LREAL(lrCounterEnergyT1_Consumption)) THEN stDataPvOut.lrCounterEnergyT1_Consumption := LINT_TO_LREAL(LREAL_TO_LINT((lrCounterEnergyT1_Consumption / 1000) * 100)) / 100; END_IF
			IF IsFinite(F_LREAL(lrCounterEnergyT2_Consumption)) THEN stDataPvOut.lrCounterEnergyT2_Consumption := LINT_TO_LREAL(LREAL_TO_LINT((lrCounterEnergyT2_Consumption / 1000) * 100)) / 100; END_IF
				IF IsFinite(F_LREAL(lrCounterEnergyT1_Production)) THEN stDataPvOut.lrCounterEnergyT1_Production := LINT_TO_LREAL(LREAL_TO_LINT((lrCounterEnergyT1_Production / 1000) * 100)) / 100; END_IF
					IF IsFinite(F_LREAL(lrCounterEnergyT2_Production)) THEN stDataPvOut.lrCounterEnergyT2_Production := LINT_TO_LREAL(LREAL_TO_LINT((lrCounterEnergyT2_Production / 1000) * 100)) / 100; END_IF
						IF IsFinite(F_LREAL(lrTotalCounterEnergy_Consumption)) THEN stDataPvOut.lrTotalCounterEnergy_Consumption := LINT_TO_LREAL(LREAL_TO_LINT((lrTotalCounterEnergy_Consumption / 1000) * 100)) / 100; END_IF
							IF IsFinite(F_LREAL(lrTotalCounterEnergy_Production)) THEN stDataPvOut.lrTotalCounterEnergy_Production := LINT_TO_LREAL(LREAL_TO_LINT((lrTotalCounterEnergy_Production / 1000) * 100)) / 100; END_IF 
					
		IF stDataPvOut.lrPower > 0 THEN
				stDataPvOut.lrPowerProduction := stDataPvOut.lrPower;
				stDataPvOut.lrPowerConsumption := 0;
		ELSIF stDataPvOut.lrPower < 0 THEN
				stDataPvOut.lrPowerProduction := 0;
				stDataPvOut.lrPowerConsumption := (stDataPvOut.lrPower * - 1);
		ELSIF stDataPvOut.lrPower = 0 THEN
				stDataPvOut.lrPowerProduction := 0;
				stDataPvOut.lrPowerConsumption := 0;
		END_IF															
ELSE																	
	stDataPvOut.lrPower := 0;
		stDataPvOut.lrCounterEnergyT1_Consumption := 0;
			stDataPvOut.lrCounterEnergyT2_Consumption := 0;
				stDataPvOut.lrCounterEnergyT1_Production := 0;
					stDataPvOut.lrCounterEnergyT2_Production := 0;
						stDataPvOut.lrPowerProduction := 0;
							stDataPvOut.lrPowerConsumption := 0;
								stDataPvOut.lrTotalCounterEnergy_Consumption := 0;
									stDataPvOut.lrTotalCounterEnergy_Production := 0;
END_IF	

(*---------------------------------------------------------------Error and Warning-------------------------------------------------------------------------------*)

stDataPvOut.byErrorWarning := 0;
	IF bWarning THEN stDataPvOut.byErrorWarning := 1; END_IF  
	IF bError THEN stDataPvOut.byErrorWarning := 2;	END_IF

//Messages and Error Codes
IF stDataPvOut.byErrorWarning = 1 AND iWarningCode = 0 THEN stDataPvOut.eMessage := E_Message_PV.eNoConnectionToBackend; 
ELSIF stDataPvOut.byErrorWarning = 2 AND iErrorCode = 0 THEN stDataPvOut.eMessage := E_Message_PV.ePvError;
ELSIF stDataPvOut.byErrorWarning = 2 AND iErrorCode = 1 THEN stDataPvOut.eMessage := E_Message_PV.eTooMuchPV;
ELSE stDataPvOut.eMessage := E_Message_PV.eNoMessage; 
END_IF

(*---------------------------------------------------------------Outputs-------------------------------------------------------------------------------*)

//Write with Delay or without
IF (bWriteWithDelay AND (timDelayOutputs.Q OR FPEnable.Q OR FNEnable.Q)) OR NOT bWriteWithDelay THEN
	stDataPvOutDelay := stDataPvOut; 
END_IF

END_FUNCTION_BLOCK

// ---- Energy/FBs Internal/Valve Control/FB_Valve_Control.TcPOU
{attribute 'hide_all_locals'}
{attribute 'conditionalshow'}
FUNCTION_BLOCK FB_Valve_Control
VAR_INPUT
	{attribute 'hide'}
	bEnable								: BOOL;							//Enable or dissable the function
	{attribute 'hide'}
	bWriteWithDelay						: BOOL;							//Write with Delay the Data to the output (Not al Output Data is writen with Delay)
	{attribute 'hide'}
	bWorkOnlyLocal						: BOOL;							//When this flag is true then the valve control work only local without the Backend commands
	{attribute 'hide'}
	rActualRoomTemperature				: REAL;							//Actual Room Temperature
	{attribute 'hide'}
	bError								: BOOL;							//Error from the Valve Control
	{attribute 'hide'}
	bWarning							: BOOL;							//Warning from the Valve Control
	{attribute 'hide'}
	iErrorCode							: INT;							//Error Code
	{attribute 'hide'}
	iWarningCode						: INT;							//Warning Code
	{attribute 'hide'}
	tTimDelayOutput						: TIME := T#5S;					//Delay Time to write some Data to the Output						
	//Data from the Lynus optimization to control the valve with the backend commands
	{attribute 'hide'}
	byMPCReady							: BYTE;							//Shows if the MPC service is ready or not.
	{attribute 'hide'}
	byNewValvePosition					: BYTE;							//The new valve positon from the Lynus Backend Service
	{attribute 'hide'}
	rNewSetTemperature					: REAL;							//Here we can set the new Set Temperatur on witch the Valve is switching on and off
	{attribute 'hide'}
	rHeartbeat							: REAL;							//Heartberat from the Service
END_VAR
VAR_OUTPUT
	{attribute 'hide'}
	stDataValveControlOut				: ST_Valve_Control_Output;		//Valve Control output data
	{attribute 'hide'}
	stDataValveControlOutDelay			: ST_Valve_Control_Output;		//Valve Control output data with delay
END_VAR
VAR
	timHB								: TON;							//Timer to check the hearbeat signal from MPC
	timDelayOutputs						: TON;							//Timer to send Data with Delay to the outputs
	timError							: TON;							//Timer for the Erro flag to set the Error with Delay
	FPEnable							: R_TRIG;						//Internal positive Edge
	FNEnable							: F_TRIG;						//Internal negative Edge
	bControllLocal						: BOOL;							//True when the Backend Service has a Error or a Warning and the Valve is controled localy
	bMPCActive							: BOOL;							//Indicates whether the new valve position is controlled by the MPC controller or whether it is controlled locally.	
	rLocalSetTemperature				: REAL := 20;					//Local Set Temperture
	rHeartbeatCP						: REAL;							//Heartbeat value to compare ols with new value
END_VAR

//Creator : Kai Ebensperger
//Company : Lynus AG
//Date : 17.03.2021
//Version : 1.0.0.0

//With this Function is possible to control a digital valve with a output from a plc
//At the moment this function controlls only digital valves
//This function can be used mainly to control floor heating valves or radiator valves.
//This Function is optimizied to work also with the Lynus Backen Service and can handle the commands from this Service
//If we have no connection to the Backend Service, then the Set temperature is set automatically to 20 °C and works locally
//Otherwise the Backend Service controll directly the valve output
//This function has also the possibility to control only local with the target setpoint and the actual room temperature.

(*---------------------------------------------------------------Limits-------------------------------------------------------------------------------*)

rActualRoomTemperature := LIMIT(-10,rActualRoomTemperature,50);
	byMPCReady := LIMIT(0,byMPCReady,1);
		byNewValvePosition := LIMIT(0,byNewValvePosition,1);
			rNewSetTemperature := LIMIT(5,rNewSetTemperature,30);
				rHeartbeat := LIMIT(0,rHeartbeat,1);			

(*---------------------------------------------------------------Enable-------------------------------------------------------------------------------*)

stDataValveControlOut.bEnabled := bEnable;				

(*---------------------------------------------------------------Error and Waring-------------------------------------------------------------------------------*)
	
timError(IN:= bError, PT:= T#5S, Q=> , ET=> );
			
stDataValveControlOut.byErrorWarning := 0;
	IF bWarning THEN stDataValveControlOut.byErrorWarning := 1; END_IF 
	IF timError.Q THEN stDataValveControlOut.byErrorWarning := 2; END_IF

//Messages and Error Codes
IF stDataValveControlOut.byErrorWarning = 1 AND iWarningCode = 0 THEN stDataValveControlOut.eMessage := E_Message_ValveControl.eNoConnectionToBackend;
ELSIF stDataValveControlOut.byErrorWarning = 1 AND iWarningCode = 1 THEN stDataValveControlOut.eMessage := E_Message_ValveControl.eValvePositionIsControlledLocal;
ELSIF stDataValveControlOut.byErrorWarning = 2 AND iErrorCode = 0 THEN stDataValveControlOut.eMessage := E_Message_ValveControl.eValvePositionError;
ELSIF stDataValveControlOut.byErrorWarning = 2 AND iErrorCode = 1 THEN stDataValveControlOut.eMessage := E_Message_ValveControl.eTooMuchValvePositions;
ELSIF stDataValveControlOut.byErrorWarning = 2 AND iErrorCode = 2 THEN stDataValveControlOut.eMessage := E_Message_ValveControl.eValvePositionIsControlledLocal;
ELSIF stDataValveControlOut.byErrorWarning = 2 AND iErrorCode = 3 THEN stDataValveControlOut.eMessage := E_Message_ValveControl.eTempSensorError;	
ELSE stDataValveControlOut.eMessage := E_Message_ValveControl.eNoMessage; 
END_IF

(*-----------------------------------------------------------------------------------------Logic-------------------------------------------------------------------------------------------------*)

//Check if MPC function in backend is activ and work
IF rHeartbeatCP = rHeartbeat THEN timHB.IN := TRUE; ELSE timHB.IN := FALSE; rHeartbeatCP := rHeartbeat; END_IF  
	timHB(IN:= , PT:= T#130S, Q=> , ET=> );	 	 

//Warning, when the Backend Service is not available
IF stDataValveControlOut.byErrorWarning = 1 AND stDataValveControlOut.eMessage = E_Message_ValveControl.eValvePositionIsControlledLocal OR 
	stDataValveControlOut.byErrorWarning = 2 AND stDataValveControlOut.eMessage = E_Message_ValveControl.eValvePositionIsControlledLocal THEN
		bControllLocal := TRUE; 
ELSE 
		bControllLocal := FALSE; 
END_IF 
	
IF NOT timHB.Q AND NOT bControllLocal AND byMPCReady = 1 AND NOT bWorkOnlyLocal THEN bMPCActive := TRUE; ELSE bMPCActive := FALSE; END_IF   

//Target Temperature from MPC
IF NOT bWorkOnlyLocal THEN
	IF NOT timHB.Q THEN
		rLocalSetTemperature := rNewSetTemperature; 
	END_IF
		//Set Temperatur to 20°C when the connection is lost to the backend system
		IF timHB.Q THEN rLocalSetTemperature := 20; END_IF 
END_IF
	
//Outputs from MPC to PLC
IF bMPCActive THEN
	//Too the Outputs from the PLC when the MPC is ok
	IF byNewValvePosition = 1 THEN 
		stDataValveControlOut.bValvePos := TRUE;
	ELSE
		stDataValveControlOut.bValvePos := FALSE;
	END_IF
END_IF

//Work only local
IF bWorkOnlyLocal THEN
	rLocalSetTemperature := rNewSetTemperature;	
END_IF

//Control the valve local with the plc if the mpc is not working
IF NOT bMPCActive THEN
	//On
	IF rActualRoomTemperature <= (rLocalSetTemperature - 0.5) THEN stDataValveControlOut.bValvePos := TRUE; END_IF  
	//Off 
	IF rActualRoomTemperature >= (rLocalSetTemperature + 0.5) THEN stDataValveControlOut.bValvePos := FALSE; END_IF	
END_IF  

//Dissable the Valve controling
IF stDataValveControlOut.byErrorWarning = 2 AND iErrorCode <> 2 OR NOT stDataValveControlOut.bEnabled THEN stDataValveControlOut.bValvePos := FALSE; END_IF  

(*---------------------------------------------------------------Outputs-------------------------------------------------------------------------------*)

timDelayOutputs(IN:= bWriteWithDelay AND bEnable AND NOT timDelayOutputs.Q, PT:= tTimDelayOutput, Q=> , ET=> );
	FPEnable(CLK:= bEnable, Q=> );
		FNEnable(CLK:= bEnable, Q=> );
		
//Write with Delay or without
IF (bWriteWithDelay AND (timDelayOutputs.Q OR FPEnable.Q OR FNEnable.Q)) OR NOT bWriteWithDelay THEN
	stDataValveControlOutDelay := stDataValveControlOut;
END_IF

END_FUNCTION_BLOCK

// ---- General/FBs Internal/Convert/BOOL/FB_CV_BOOL_TO_WORD.TcPOU
{attribute 'conditionalshow'}
FUNCTION_BLOCK FB_CV_BOOL_TO_WORD
VAR_INPUT
	{attribute 'hide'}
	arrInputValue			: ARRAY[0..15] OF BOOL;				//Input value that is converted into the output value
END_VAR
VAR_OUTPUT
	{attribute 'hide'}
	wOutputValue			: WORD;								//Converted output value
END_VAR
VAR
END_VAR

//Creator : Kai Ebensperger
//Company : Lynus AG
//Date : 28.04.2021
//Version : 1.0.0.0

//With this functionblock its possible to convert a certain Datatyp in a other Datatype
//BOOL TO WORD
//Created for the Edge Device Lib over Modbus TCP
//Modbus TCP is WORD oriented

wOutputValue.0 := arrInputValue[0];
wOutputValue.1 := arrInputValue[1];
wOutputValue.2 := arrInputValue[2];
wOutputValue.3 := arrInputValue[3];
wOutputValue.4 := arrInputValue[4];
wOutputValue.5 := arrInputValue[5];
wOutputValue.6 := arrInputValue[6];
wOutputValue.7 := arrInputValue[7];
wOutputValue.8 := arrInputValue[8];
wOutputValue.9 := arrInputValue[9];
wOutputValue.10 := arrInputValue[10];
wOutputValue.11 := arrInputValue[11];
wOutputValue.12 := arrInputValue[12];
wOutputValue.13 := arrInputValue[13];
wOutputValue.14 := arrInputValue[14];
wOutputValue.15 := arrInputValue[15];

END_FUNCTION_BLOCK

// ---- General/FBs Internal/Convert/BOOL/FB_CV_WORD_TO_BOOL.TcPOU
{attribute 'conditionalshow'}
FUNCTION_BLOCK FB_CV_WORD_TO_BOOL
VAR_INPUT
	{attribute 'hide'}
	wInputValue			: WORD;								//Input value that is converted into the output value
END_VAR
VAR_OUTPUT
	{attribute 'hide'}
	arrOutputValue		: ARRAY[0..15] OF BOOL;				//Converted output value
END_VAR
VAR
END_VAR

//Creator : Kai Ebensperger
//Company : Lynus AG
//Date : 28.04.2021
//Version : 1.0.0.0

//With this functionblock its possible to convert a certain Datatyp in a other Datatype
//WORD TO BOOL
//Created for the Edge Device Lib over Modbus TCP
//Modbus TCP is WORD oriented

arrOutputValue[0] := wInputValue.0;
arrOutputValue[1] := wInputValue.1;
arrOutputValue[2] := wInputValue.2;
arrOutputValue[3] := wInputValue.3;
arrOutputValue[4] := wInputValue.4;
arrOutputValue[5] := wInputValue.5;
arrOutputValue[6] := wInputValue.6;
arrOutputValue[7] := wInputValue.7;
arrOutputValue[8] := wInputValue.8;
arrOutputValue[9] := wInputValue.9;
arrOutputValue[10] := wInputValue.10;
arrOutputValue[11] := wInputValue.11;
arrOutputValue[12] := wInputValue.12;
arrOutputValue[13] := wInputValue.13;
arrOutputValue[14] := wInputValue.14;
arrOutputValue[15] := wInputValue.15;

END_FUNCTION_BLOCK

// ---- General/FBs Internal/Convert/BYTE/FB_CV_BYTE_TO_WORD.TcPOU
{attribute 'conditionalshow'}
FUNCTION_BLOCK FB_CV_BYTE_TO_WORD
VAR_INPUT
	{attribute 'hide'}
	byInputValue_1					: BYTE;								//Input value that is converted into the output value	
	{attribute 'hide'}						
	byInputValue_2					: BYTE;								//Input value that is converted into the output value
	{attribute 'hide'}
	eByteOrderForConvert			: eByteOrder;						//Byte Format
END_VAR
VAR_OUTPUT
	{attribute 'hide'}
	wOutputValue					: WORD;								//Converted output value
END_VAR
VAR
END_VAR

//Creator : Kai Ebensperger
//Company : Lynus AG
//Date : 28.04.2021
//Version : 1.0.0.0

//With this functionblock its possible to convert a certain Datatyp in a other Datatype
//The byte order can be selected between BigEndian and LittleEndian
//BYTE TO WORD
//Created for the Edge Device Lib over Modbus TCP
//Modbus TCP is WORD oriented

IF eByteOrderForConvert = eByteOrder.eBigEndian THEN
	wOutputValue := SHL(BYTE_TO_WORD(byInputValue_1),8) + BYTE_TO_WORD(byInputValue_2);
ELSE
	wOutputValue := SHL(BYTE_TO_WORD(byInputValue_2),8) + BYTE_TO_WORD(byInputValue_1);
END_IF

END_FUNCTION_BLOCK

// ---- General/FBs Internal/Convert/BYTE/FB_CV_WORD_TO_BYTE.TcPOU
{attribute 'conditionalshow'}
FUNCTION_BLOCK FB_CV_WORD_TO_BYTE
VAR_INPUT
	{attribute 'hide'}
	wInputValue						: WORD;								//Input value that is converted into the output value
	{attribute 'hide'}
	eByteOrderForConvert			: eByteOrder;						//Byte Format
END_VAR
VAR_OUTPUT
	{attribute 'hide'}
	byOutputValue_1					: BYTE;								//Converted output value	
	{attribute 'hide'}						
	byOutputValue_2					: BYTE;								//Converted output value
END_VAR
VAR
END_VAR

//Creator : Kai Ebensperger
//Company : Lynus AG
//Date : 28.04.2021
//Version : 1.0.0.0

//With this functionblock its possible to convert a certain Datatyp in a other Datatype
//The byte order can be selected between BigEndian and LittleEndian
//WORD TO BYTE
//Created for the Edge Device Lib over Modbus TCP
//Modbus TCP is WORD oriented

IF eByteOrderForConvert = eByteOrder.eBigEndian THEN
	byOutputValue_1 := WORD_TO_BYTE(SHR(wInputValue,8) AND 16#FFFF);
	byOutputValue_2 := WORD_TO_BYTE(wInputValue AND 16#FFFF);
ELSE
	byOutputValue_2 := WORD_TO_BYTE(SHR(wInputValue,8) AND 16#FFFF);
	byOutputValue_1 := WORD_TO_BYTE(wInputValue AND 16#FFFF);
END_IF

END_FUNCTION_BLOCK

// ---- General/FBs Internal/Convert/DINT/FB_CV_DINT_TO_WORD.TcPOU
{attribute 'conditionalshow'}
FUNCTION_BLOCK FB_CV_DINT_TO_WORD
VAR_INPUT
	{attribute 'hide'}
	diInputValue				: DINT;								//Input value that is converted into the output value
	{attribute 'hide'}
	eByteOrderForConvert		: eByteOrder;						//Byte Format							
END_VAR
VAR_OUTPUT
	{attribute 'hide'}
	wOutputValue_1				: WORD;								//Converted output value
	{attribute 'hide'}
	wOutputValue_2				: WORD;								//Converted output value
END_VAR
VAR
END_VAR

//Creator : Kai Ebensperger
//Company : Lynus AG
//Date : 28.04.2021
//Version : 1.0.0.0

//With this functionblock its possible to convert a certain Datatyp in a other Datatype
//The byte order can be selected between BigEndian and LittleEndian
//DINT TO WORD
//Created for the Edge Device Lib over Modbus TCP
//Modbus TCP is WORD oriented

IF eByteOrderForConvert = eByteOrder.eBigEndian THEN
	wOutputValue_1 := DWORD_TO_WORD(SHR(DINT_TO_DWORD(diInputValue),16) AND 16#FFFF);
	wOutputValue_2 := DWORD_TO_WORD(DINT_TO_DWORD(diInputValue)) AND 16#FFFF;
ELSE
	wOutputValue_2 := DWORD_TO_WORD(SHR(DINT_TO_DWORD(diInputValue),16) AND 16#FFFF);
	wOutputValue_1 := DWORD_TO_WORD(DINT_TO_DWORD(diInputValue)) AND 16#FFFF;
END_IF

END_FUNCTION_BLOCK

// ---- General/FBs Internal/Convert/DINT/FB_CV_WORD_TO_DINT.TcPOU
{attribute 'conditionalshow'}
FUNCTION_BLOCK FB_CV_WORD_TO_DINT
VAR_INPUT
	{attribute 'hide'}
	wInputValue_1				: WORD;								//Input value that is converted into the output value
	{attribute 'hide'}
	wInputValue_2				: WORD;								//Input value that is converted into the output value
	{attribute 'hide'}
	eByteOrderForConvert		: eByteOrder;						//Byte Format
END_VAR
VAR_OUTPUT
	{attribute 'hide'}
	diOutputValue				: DINT;								//Converted output value							
END_VAR
VAR
END_VAR

//Creator : Kai Ebensperger
//Company : Lynus AG
//Date : 28.04.2021
//Version : 1.0.0.0

//With this functionblock its possible to convert a certain Datatyp in a other Datatype
//The byte order can be selected between BigEndian and LittleEndian
//WORD TO DINT
//Created for the Edge Device Lib over Modbus TCP
//Modbus TCP is WORD oriented

IF eByteOrderForConvert = eByteOrder.eBigEndian THEN
	diOutputValue := DWORD_TO_DINT(SHL(WORD_TO_DWORD(wInputValue_1),16) + WORD_TO_DWORD(wInputValue_2));
ELSE
	diOutputValue := DWORD_TO_DINT(SHL(WORD_TO_DWORD(wInputValue_2),16) + WORD_TO_DWORD(wInputValue_1));
END_IF

END_FUNCTION_BLOCK

// ---- General/FBs Internal/Convert/DWORD/FB_CV_DWORD_TO_WORD.TcPOU
{attribute 'conditionalshow'}
FUNCTION_BLOCK FB_CV_DWORD_TO_WORD
VAR_INPUT
	{attribute 'hide'}
	dwInputValue				: DWORD;							//Input value that is converted into the output value	
	{attribute 'hide'}						
	eByteOrderForConvert		: eByteOrder;						//Byte Format
END_VAR
VAR_OUTPUT
	{attribute 'hide'}
	wOutputValue_1				: WORD;								//Converted output value
	{attribute 'hide'}
	wOutputValue_2				: WORD;								//Converted output value
END_VAR
VAR
END_VAR

//Creator : Kai Ebensperger
//Company : Lynus AG
//Date : 28.04.2021
//Version : 1.0.0.0

//With this functionblock its possible to convert a certain Datatyp in a other Datatype
//The byte order can be selected between BigEndian and LittleEndian
//DWORD TO WORD
//Created for the Edge Device Lib over Modbus TCP
//Modbus TCP is WORD oriented

IF eByteOrderForConvert = eByteOrder.eBigEndian THEN
	wOutputValue_1 := DWORD_TO_WORD(SHR(dwInputValue,16) AND 16#FFFF);
	wOutputValue_2 := DWORD_TO_WORD(dwInputValue) AND 16#FFFF;
ELSE
	wOutputValue_2 := DWORD_TO_WORD(SHR(dwInputValue,16) AND 16#FFFF);
	wOutputValue_1 := DWORD_TO_WORD(dwInputValue) AND 16#FFFF;
END_IF

END_FUNCTION_BLOCK

// ---- General/FBs Internal/Convert/DWORD/FB_CV_WORD_TO_DWORD.TcPOU
{attribute 'conditionalshow'}
FUNCTION_BLOCK FB_CV_WORD_TO_DWORD
VAR_INPUT
	{attribute 'hide'}
	wInputValue_1				: WORD;								//Input value that is converted into the output value
	{attribute 'hide'}
	wInputValue_2				: WORD;								//Input value that is converted into the output value
	{attribute 'hide'}
	eByteOrderForConvert		: eByteOrder;						//Byte Format
END_VAR
VAR_OUTPUT
	{attribute 'hide'}
	dwOutputValue				: DWORD;							//Converted output value							
END_VAR
VAR
END_VAR

//Creator : Kai Ebensperger
//Company : Lynus AG
//Date : 28.04.2021
//Version : 1.0.0.0

//With this functionblock its possible to convert a certain Datatyp in a other Datatype
//The byte order can be selected between BigEndian and LittleEndian
//WORD TO DWORD
//Created for the Edge Device Lib over Modbus TCP
//Modbus TCP is WORD oriented

IF eByteOrderForConvert = eByteOrder.eBigEndian THEN
	dwOutputValue := SHL(WORD_TO_DWORD(wInputValue_1),16) + WORD_TO_DWORD(wInputValue_2);
ELSE
	dwOutputValue := SHL(WORD_TO_DWORD(wInputValue_2),16) + WORD_TO_DWORD(wInputValue_1);
END_IF

END_FUNCTION_BLOCK

// ---- General/FBs Internal/Convert/INT/FB_CV_INT_TO_WORD.TcPOU
{attribute 'conditionalshow'}
FUNCTION_BLOCK FB_CV_INT_TO_WORD
VAR_INPUT
	{attribute 'hide'}
	iInputValue					: INT;								//Input value that is converted into the output value							
END_VAR
VAR_OUTPUT
	{attribute 'hide'}
	wOutputValue				: WORD;								//Converted output value
END_VAR
VAR
END_VAR

//Creator : Kai Ebensperger
//Company : Lynus AG
//Date : 28.04.2021
//Version : 1.0.0.0

//With this functionblock its possible to convert a certain Datatyp in a other Datatype
//INT TO WORD
//Created for the Edge Device Lib over Modbus TCP
//Modbus TCP is WORD oriented

wOutputValue := INT_TO_WORD(iInputValue);

END_FUNCTION_BLOCK

// ---- General/FBs Internal/Convert/INT/FB_CV_WORD_TO_INT.TcPOU
{attribute 'conditionalshow'}
FUNCTION_BLOCK FB_CV_WORD_TO_INT
VAR_INPUT
	{attribute 'hide'}
	wInputValue					: WORD;								//Input value that is converted into the output value
END_VAR
VAR_OUTPUT
	{attribute 'hide'}
	iOutputValue				: INT;								//Converted output value							
END_VAR
VAR
END_VAR

//Creator : Kai Ebensperger
//Company : Lynus AG
//Date : 28.04.2021
//Version : 1.0.0.0

//With this functionblock its possible to convert a certain Datatyp in a other Datatype
//WORD TO INT
//Created for the Edge Device Lib over Modbus TCP
//Modbus TCP is WORD oriented

iOutputValue := WORD_TO_INT(wInputValue);

END_FUNCTION_BLOCK

// ---- General/FBs Internal/Convert/LINT/FB_CV_LINT_TO_WORD.TcPOU
{attribute 'conditionalshow'}
FUNCTION_BLOCK FB_CV_LINT_TO_WORD
VAR_INPUT
	{attribute 'hide'}
	liInputValue				: LINT;								//Input value that is converted into the output value
	{attribute 'hide'}
	eByteOrderForConvert		: eByteOrder;						//Byte Format							
END_VAR
VAR_OUTPUT
	{attribute 'hide'}
	wOutputValue_1				: WORD;								//Converted output value
	{attribute 'hide'}
	wOutputValue_2				: WORD;								//Converted output value
	{attribute 'hide'}
	wOutputValue_3				: WORD;								//Converted output value
	{attribute 'hide'}
	wOutputValue_4				: WORD;								//Converted output value
END_VAR
VAR
END_VAR

//Creator : Kai Ebensperger
//Company : Lynus AG
//Date : 28.04.2021
//Version : 1.0.0.0

//With this functionblock its possible to convert a certain Datatyp in a other Datatype
//The byte order can be selected between BigEndian and LittleEndian
//LINT TO WORD
//Created for the Edge Device Lib over Modbus TCP
//Modbus TCP is WORD oriented

IF eByteOrderForConvert = eByteOrder.eBigEndian THEN
	wOutputValue_1 := ULINT_TO_WORD(SHR(LINT_TO_ULINT(liInputValue),48) AND 16#FFFF);
	wOutputValue_2 := ULINT_TO_WORD(SHR(LINT_TO_ULINT(liInputValue),32) AND 16#FFFF);
	wOutputValue_3 := ULINT_TO_WORD(SHR(LINT_TO_ULINT(liInputValue),16) AND 16#FFFF);
	wOutputValue_4 := ULINT_TO_WORD(LINT_TO_ULINT(liInputValue)) AND 16#FFFF;
ELSE
	wOutputValue_4 := ULINT_TO_WORD(SHR(LINT_TO_ULINT(liInputValue),48) AND 16#FFFF);
	wOutputValue_3 := ULINT_TO_WORD(SHR(LINT_TO_ULINT(liInputValue),32) AND 16#FFFF);
	wOutputValue_2 := ULINT_TO_WORD(SHR(LINT_TO_ULINT(liInputValue),16) AND 16#FFFF);
	wOutputValue_1 := ULINT_TO_WORD(LINT_TO_ULINT(liInputValue)) AND 16#FFFF;
END_IF

END_FUNCTION_BLOCK

// ---- General/FBs Internal/Convert/LINT/FB_CV_WORD_TO_LINT.TcPOU
{attribute 'conditionalshow'}
FUNCTION_BLOCK FB_CV_WORD_TO_LINT
VAR_INPUT
	{attribute 'hide'}
	wInputValue_1				: WORD;								//Input value that is converted into the output value
	{attribute 'hide'}
	wInputValue_2				: WORD;								//Input value that is converted into the output value
	{attribute 'hide'}
	wInputValue_3				: WORD;								//Input value that is converted into the output value
	{attribute 'hide'}
	wInputValue_4				: WORD;								//Input value that is converted into the output value
	{attribute 'hide'}
	eByteOrderForConvert		: eByteOrder;						//Byte Format
END_VAR
VAR_OUTPUT
	{attribute 'hide'}
	liOutputValue				: LINT;								//Converted output value							
END_VAR
VAR
END_VAR

//Creator : Kai Ebensperger
//Company : Lynus AG
//Date : 28.04.2021
//Version : 1.0.0.0

//With this functionblock its possible to convert a certain Datatyp in a other Datatype
//The byte order can be selected between BigEndian and LittleEndian
//WORD TO LINT
//Created for the Edge Device Lib over Modbus TCP
//Modbus TCP is WORD oriented

IF eByteOrderForConvert = eByteOrder.eBigEndian THEN
	liOutputValue := ULINT_TO_LINT(SHL(WORD_TO_ULINT(wInputValue_1),48) + SHL(WORD_TO_ULINT(wInputValue_2),32) + SHL(WORD_TO_ULINT(wInputValue_3),16) + WORD_TO_DWORD(wInputValue_4));
ELSE
	liOutputValue := ULINT_TO_LINT(SHL(WORD_TO_ULINT(wInputValue_4),48) + SHL(WORD_TO_ULINT(wInputValue_3),32) + SHL(WORD_TO_ULINT(wInputValue_2),16) + WORD_TO_DWORD(wInputValue_1));
END_IF

END_FUNCTION_BLOCK

// ---- General/FBs Internal/Convert/LREAL_FLOAT/FB_CV_LREAL_FLOAT_TO_WORD.TcPOU
{attribute 'hide_all_locals'}
{attribute 'conditionalshow'}
FUNCTION_BLOCK FB_CV_LREAL_FLOAT_TO_WORD
VAR_INPUT
	{attribute 'hide'}
	lrInputValue				: LREAL;							//Input value that is converted into the output value
	{attribute 'hide'}							
	eByteOrderForConvert		: eByteOrder;						//Byte Format
END_VAR
VAR_OUTPUT
	{attribute 'hide'}
	wOutputValue_1				: WORD;								//Converted output value
	{attribute 'hide'}
	wOutputValue_2				: WORD;								//Converted output value
	{attribute 'hide'}
	wOutputValue_3				: WORD;								//Converted output value
	{attribute 'hide'}
	wOutputValue_4				: WORD;								//Converted output value
END_VAR
VAR
	unConvertLRealToULINT		: ST_UN_FLOAT_CONVERT_ULINT_LREAL;	//Union to convert the value
END_VAR

//Creator : Kai Ebensperger
//Company : Lynus AG
//Date : 28.04.2021
//Version : 1.0.0.0

//With this functionblock its possible to convert a certain Datatyp in a other Datatype
//The byte order can be selected between BigEndian and LittleEndian
//LREAL TO WORD
//Created for the Edge Device Lib over Modbus TCP
//Modbus TCP is WORD oriented

unConvertLRealToULINT.lrValueFloat := lrInputValue;

IF eByteOrderForConvert = eByteOrder.eBigEndian THEN
	wOutputValue_1 := ULINT_TO_WORD(SHR(unConvertLRealToULINT.uliRawValue,48) AND 16#FFFF);
	wOutputValue_2 := ULINT_TO_WORD(SHR(unConvertLRealToULINT.uliRawValue,32) AND 16#FFFF);
	wOutputValue_3 := ULINT_TO_WORD(SHR(unConvertLRealToULINT.uliRawValue,16) AND 16#FFFF);
	wOutputValue_4 := ULINT_TO_WORD(unConvertLRealToULINT.uliRawValue) AND 16#FFFF;
ELSE
	wOutputValue_4 := ULINT_TO_WORD(SHR(unConvertLRealToULINT.uliRawValue,48) AND 16#FFFF);
	wOutputValue_3 := ULINT_TO_WORD(SHR(unConvertLRealToULINT.uliRawValue,32) AND 16#FFFF);
	wOutputValue_2 := ULINT_TO_WORD(SHR(unConvertLRealToULINT.uliRawValue,16) AND 16#FFFF);
	wOutputValue_1 := ULINT_TO_WORD(unConvertLRealToULINT.uliRawValue) AND 16#FFFF;
END_IF

END_FUNCTION_BLOCK

// ---- General/FBs Internal/Convert/LREAL_FLOAT/FB_CV_WORD_TO_LREAL_FLOAT.TcPOU
{attribute 'hide_all_locals'}
{attribute 'conditionalshow'}
FUNCTION_BLOCK FB_CV_WORD_TO_LREAL_FLOAT
VAR_INPUT
	{attribute 'hide'}
	wInputValue_1				: WORD;								//Input value that is converted into the output value
	{attribute 'hide'}
	wInputValue_2				: WORD;								//Input value that is converted into the output value
	{attribute 'hide'}
	wInputValue_3				: WORD;								//Input value that is converted into the output value
	{attribute 'hide'}
	wInputValue_4				: WORD;								//Input value that is converted into the output value
	{attribute 'hide'}
	eByteOrderForConvert		: eByteOrder;						//Byte Format
END_VAR
VAR_OUTPUT
	{attribute 'hide'}
	lrOutputValue				: LREAL;							//Converted output value							
END_VAR
VAR
	unConvertLRealToULINT		: ST_UN_FLOAT_CONVERT_ULINT_LREAL;	//Union to convert the value
END_VAR

//Creator : Kai Ebensperger
//Company : Lynus AG
//Date : 28.04.2021
//Version : 1.0.0.0

//With this functionblock its possible to convert a certain Datatyp in a other Datatype
//The byte order can be selected between BigEndian and LittleEndian
//WORD TO LREAL
//Created for the Edge Device Lib over Modbus TCP
//Modbus TCP is WORD oriented

IF eByteOrderForConvert = eByteOrder.eBigEndian THEN
	unConvertLRealToULINT.uliRawValue := SHL(WORD_TO_ULINT(wInputValue_1),48) + SHL(WORD_TO_ULINT(wInputValue_2),32) + SHL(WORD_TO_ULINT(wInputValue_3),16) + WORD_TO_DWORD(wInputValue_4);
ELSE
	unConvertLRealToULINT.uliRawValue := SHL(WORD_TO_ULINT(wInputValue_4),48) + SHL(WORD_TO_ULINT(wInputValue_3),32) + SHL(WORD_TO_ULINT(wInputValue_2),16) + WORD_TO_DWORD(wInputValue_1);
END_IF

IF IsFinite(F_LREAL(unConvertLRealToULINT.lrValueFloat)) THEN
	lrOutputValue := unConvertLRealToULINT.lrValueFloat;
END_IF

END_FUNCTION_BLOCK

// ---- General/FBs Internal/Convert/LWORD/FB_CV_LWORD_TO_WORD.TcPOU
{attribute 'conditionalshow'}
FUNCTION_BLOCK FB_CV_LWORD_TO_WORD
VAR_INPUT
	{attribute 'hide'}
	lwInputValue				: LWORD;							//Input value that is converted into the output value	
	{attribute 'hide'}						
	eByteOrderForConvert		: eByteOrder;						//Byte Format
END_VAR
VAR_OUTPUT
	{attribute 'hide'}
	wOutputValue_1				: WORD;								//Converted output value
	{attribute 'hide'}
	wOutputValue_2				: WORD;								//Converted output value
	{attribute 'hide'}
	wOutputValue_3				: WORD;								//Converted output value
	{attribute 'hide'}
	wOutputValue_4				: WORD;								//Converted output value
END_VAR
VAR
END_VAR

//Creator : Kai Ebensperger
//Company : Lynus AG
//Date : 28.04.2021
//Version : 1.0.0.0

//With this functionblock its possible to convert a certain Datatyp in a other Datatype
//The byte order can be selected between BigEndian and LittleEndian
//LWORD TO WORD
//Created for the Edge Device Lib over Modbus TCP
//Modbus TCP is WORD oriented

IF eByteOrderForConvert = eByteOrder.eBigEndian THEN
	wOutputValue_1 := LWORD_TO_WORD(SHR(lwInputValue,48) AND 16#FFFF);
	wOutputValue_2 := LWORD_TO_WORD(SHR(lwInputValue,32) AND 16#FFFF);
	wOutputValue_3 := LWORD_TO_WORD(SHR(lwInputValue,16) AND 16#FFFF);
	wOutputValue_4 := LWORD_TO_WORD(lwInputValue) AND 16#FFFF;
ELSE
	wOutputValue_4 := LWORD_TO_WORD(SHR(lwInputValue,48) AND 16#FFFF);
	wOutputValue_3 := LWORD_TO_WORD(SHR(lwInputValue,32) AND 16#FFFF);
	wOutputValue_2 := LWORD_TO_WORD(SHR(lwInputValue,16) AND 16#FFFF);
	wOutputValue_1 := LWORD_TO_WORD(lwInputValue) AND 16#FFFF;
END_IF

END_FUNCTION_BLOCK

// ---- General/FBs Internal/Convert/LWORD/FB_CV_WORD_TO_LWORD.TcPOU
{attribute 'conditionalshow'}
FUNCTION_BLOCK FB_CV_WORD_TO_LWORD
VAR_INPUT
	{attribute 'hide'}
	wInputValue_1				: WORD;								//Input value that is converted into the output value
	{attribute 'hide'}
	wInputValue_2				: WORD;								//Input value that is converted into the output value
	{attribute 'hide'}
	wInputValue_3				: WORD;								//Input value that is converted into the output value
	{attribute 'hide'}
	wInputValue_4				: WORD;								//Input value that is converted into the output value
	{attribute 'hide'}
	eByteOrderForConvert		: eByteOrder;						//Byte Format
END_VAR
VAR_OUTPUT
	{attribute 'hide'}
	lwOutputValue				: LWORD;							//Converted output value							
END_VAR
VAR
END_VAR

//Creator : Kai Ebensperger
//Company : Lynus AG
//Date : 28.04.2021
//Version : 1.0.0.0

//With this functionblock its possible to convert a certain Datatyp in a other Datatype
//The byte order can be selected between BigEndian and LittleEndian
//WORD TO LWORD
//Created for the Edge Device Lib over Modbus TCP
//Modbus TCP is WORD oriented

IF eByteOrderForConvert = eByteOrder.eBigEndian THEN
	lwOutputValue := SHL(WORD_TO_LWORD(wInputValue_1),48) + SHL(WORD_TO_LWORD(wInputValue_2),32) + SHL(WORD_TO_LWORD(wInputValue_3),16) + WORD_TO_LWORD(wInputValue_4);
ELSE
	lwOutputValue := SHL(WORD_TO_LWORD(wInputValue_4),48) + SHL(WORD_TO_LWORD(wInputValue_3),32) + SHL(WORD_TO_LWORD(wInputValue_2),16) + WORD_TO_LWORD(wInputValue_1);
END_IF

END_FUNCTION_BLOCK

// ---- General/FBs Internal/Convert/REAL_FLOAT/FB_CV_REAL_FLOAT_TO_WORD.TcPOU
{attribute 'conditionalshow'}
{attribute 'hide_all_locals'}
FUNCTION_BLOCK FB_CV_REAL_FLOAT_TO_WORD
VAR_INPUT
	{attribute 'hide'}
	rInputValue					: REAL;								//Input value that is converted into the output value	
	{attribute 'hide'}						
	eByteOrderForConvert		: eByteOrder;						//Byte Format
END_VAR
VAR_OUTPUT
	{attribute 'hide'}
	wOutputValue_1				: WORD;								//Converted output value
	{attribute 'hide'}
	wOutputValue_2				: WORD;								//Converted output value
END_VAR
VAR
	unConvertRealToDword		: ST_UN_FLOAT_CONVERT_DWORD_REAL;	//Union to convert the value
END_VAR

//Creator : Kai Ebensperger
//Company : Lynus AG
//Date : 28.04.2021
//Version : 1.0.0.0

//With this functionblock its possible to convert a certain Datatyp in a other Datatype
//The byte order can be selected between BigEndian and LittleEndian
//REAL TO WORD
//Created for the Edge Device Lib over Modbus TCP
//Modbus TCP is WORD oriented

unConvertRealToDword.rValueFloat := rInputValue;

IF eByteOrderForConvert = eByteOrder.eBigEndian THEN
	wOutputValue_1 := DWORD_TO_WORD(SHR(unConvertRealToDword.dwRawValue,16) AND 16#FFFF);
	wOutputValue_2 := DWORD_TO_WORD(unConvertRealToDword.dwRawValue) AND 16#FFFF;
ELSE
	wOutputValue_2 := DWORD_TO_WORD(SHR(unConvertRealToDword.dwRawValue,16) AND 16#FFFF);
	wOutputValue_1 := DWORD_TO_WORD(unConvertRealToDword.dwRawValue) AND 16#FFFF;
END_IF

END_FUNCTION_BLOCK

// ---- General/FBs Internal/Convert/REAL_FLOAT/FB_CV_WORD_TO_REAL_FLOAT.TcPOU
{attribute 'conditionalshow'}
{attribute 'hide_all_locals'}
FUNCTION_BLOCK FB_CV_WORD_TO_REAL_FLOAT
VAR_INPUT
	{attribute 'hide'}
	wInputValue_1				: WORD;								//Input value that is converted into the output value
	{attribute 'hide'}
	wInputValue_2				: WORD;								//Input value that is converted into the output value
	{attribute 'hide'}
	eByteOrderForConvert		: eByteOrder;						//Byte Format
END_VAR
VAR_OUTPUT
	{attribute 'hide'}
	rOutputValue				: REAL;								//Converted output value							
END_VAR
VAR
	unConvertRealToDword		: ST_UN_FLOAT_CONVERT_DWORD_REAL;	//Union to convert the value
END_VAR

//Creator : Kai Ebensperger
//Company : Lynus AG
//Date : 28.04.2021
//Version : 1.0.0.0

//With this functionblock its possible to convert a certain Datatyp in a other Datatype
//The byte order can be selected between BigEndian and LittleEndian
//WORD TO REAL
//Created for the Edge Device Lib over Modbus TCP
//Modbus TCP is WORD oriented

IF eByteOrderForConvert = eByteOrder.eBigEndian THEN
	unConvertRealToDword.dwRawValue := SHL(WORD_TO_DWORD(wInputValue_1),16) + WORD_TO_DWORD(wInputValue_2);
ELSE
	unConvertRealToDword.dwRawValue := SHL(WORD_TO_DWORD(wInputValue_2),16) + WORD_TO_DWORD(wInputValue_1);
END_IF

IF IsFinite(F_REAL(unConvertRealToDword.rValueFloat)) THEN
	rOutputValue := unConvertRealToDword.rValueFloat;
END_IF

END_FUNCTION_BLOCK

// ---- General/FBs Internal/Convert/SINT/FB_CV_SINT_TO_WORD.TcPOU
{attribute 'conditionalshow'}
FUNCTION_BLOCK FB_CV_SINT_TO_WORD
VAR_INPUT
	{attribute 'hide'}
	siInputValue_1				: SINT;								//Input value that is converted into the output value	
	{attribute 'hide'}						
	siInputValue_2				: SINT;								//Input value that is converted into the output value
	{attribute 'hide'}
	eByteOrderForConvert		: eByteOrder;						//Byte Format
END_VAR
VAR_OUTPUT
	{attribute 'hide'}
	wOutputValue				: WORD;								//Converted output value
END_VAR
VAR
END_VAR

//Creator : Kai Ebensperger
//Company : Lynus AG
//Date : 28.04.2021
//Version : 1.0.0.0

//With this functionblock its possible to convert a certain Datatyp in a other Datatype
//The byte order can be selected between BigEndian and LittleEndian
//SINT TO WORD
//Created for the Edge Device Lib over Modbus TCP
//Modbus TCP is WORD oriented

IF eByteOrderForConvert = eByteOrder.eBigEndian THEN
	wOutputValue := SHL(BYTE_TO_WORD(SINT_TO_BYTE(siInputValue_1)),8) + BYTE_TO_WORD(SINT_TO_BYTE(siInputValue_2));
ELSE
	wOutputValue := SHL(BYTE_TO_WORD(SINT_TO_BYTE(siInputValue_2)),8) + BYTE_TO_WORD(SINT_TO_BYTE(siInputValue_1));
END_IF

END_FUNCTION_BLOCK

// ---- General/FBs Internal/Convert/SINT/FB_CV_WORD_TO_SINT.TcPOU
{attribute 'conditionalshow'}
FUNCTION_BLOCK FB_CV_WORD_TO_SINT
VAR_INPUT
	{attribute 'hide'}
	wInputValue					: WORD;								//Input value that is converted into the output value
	{attribute 'hide'}
	eByteOrderForConvert		: eByteOrder;						//Byte Format
END_VAR
VAR_OUTPUT
	{attribute 'hide'}
	siOutputValue_1				: SINT;								//Converted output value
	{attribute 'hide'}							
	siOutputValue_2				: SINT;								//Converted output value
END_VAR
VAR
END_VAR

//Creator : Kai Ebensperger
//Company : Lynus AG
//Date : 28.04.2021
//Version : 1.0.0.0

//With this functionblock its possible to convert a certain Datatyp in a other Datatype
//The byte order can be selected between BigEndian and LittleEndian
//WORD TO SINT
//Created for the Edge Device Lib over Modbus TCP
//Modbus TCP is WORD oriented

IF eByteOrderForConvert = eByteOrder.eBigEndian THEN
	siOutputValue_1 := BYTE_TO_SINT(WORD_TO_BYTE(SHR(wInputValue,8) AND 16#FFFF));
	siOutputValue_2 := BYTE_TO_SINT(WORD_TO_BYTE(wInputValue AND 16#FFFF));
ELSE
	siOutputValue_2 := BYTE_TO_SINT(WORD_TO_BYTE(SHR(wInputValue,8) AND 16#FFFF));
	siOutputValue_1 := BYTE_TO_SINT(WORD_TO_BYTE(wInputValue AND 16#FFFF));
END_IF

END_FUNCTION_BLOCK

// ---- General/FBs Internal/Convert/UDINT/FB_CV_UDINT_TO_WORD.TcPOU
{attribute 'conditionalshow'}
FUNCTION_BLOCK FB_CV_UDINT_TO_WORD
VAR_INPUT
	{attribute 'hide'}
	udiInputValue				: UDINT;							//Input value that is converted into the output value	
	{attribute 'hide'}						
	eByteOrderForConvert		: eByteOrder;						//Byte Format
END_VAR
VAR_OUTPUT
	{attribute 'hide'}
	wOutputValue_1				: WORD;								//Converted output value
	{attribute 'hide'}
	wOutputValue_2				: WORD;								//Converted output value
END_VAR
VAR
END_VAR

//Creator : Kai Ebensperger
//Company : Lynus AG
//Date : 28.04.2021
//Version : 1.0.0.0

//With this functionblock its possible to convert a certain Datatyp in a other Datatype
//The byte order can be selected between BigEndian and LittleEndian
//UDINT TO WORD
//Created for the Edge Device Lib over Modbus TCP
//Modbus TCP is WORD oriented

IF eByteOrderForConvert = eByteOrder.eBigEndian THEN
	wOutputValue_1 := UDINT_TO_WORD(SHR(udiInputValue,16) AND 16#FFFF);
	wOutputValue_2 := UDINT_TO_WORD(udiInputValue) AND 16#FFFF;
ELSE
	wOutputValue_2 := UDINT_TO_WORD(SHR(udiInputValue,16) AND 16#FFFF);
	wOutputValue_1 := UDINT_TO_WORD(udiInputValue) AND 16#FFFF;
END_IF

END_FUNCTION_BLOCK

// ---- General/FBs Internal/Convert/UDINT/FB_CV_WORD_TO_UDINT.TcPOU
{attribute 'conditionalshow'}
FUNCTION_BLOCK FB_CV_WORD_TO_UDINT
VAR_INPUT
	{attribute 'hide'}
	wInputValue_1				: WORD;								//Input value that is converted into the output value
	{attribute 'hide'}
	wInputValue_2				: WORD;								//Input value that is converted into the output value
	{attribute 'hide'}
	eByteOrderForConvert		: eByteOrder;						//Byte Format
END_VAR
VAR_OUTPUT
	{attribute 'hide'}
	udiOutputValue				: UDINT;							//Converted output value							
END_VAR
VAR
END_VAR

//Creator : Kai Ebensperger
//Company : Lynus AG
//Date : 28.04.2021
//Version : 1.0.0.0

//With this functionblock its possible to convert a certain Datatyp in a other Datatype
//The byte order can be selected between BigEndian and LittleEndian
//WORD TO UDINT
//Created for the Edge Device Lib over Modbus TCP
//Modbus TCP is WORD oriented

IF eByteOrderForConvert = eByteOrder.eBigEndian THEN
	udiOutputValue := SHL(WORD_TO_UDINT(wInputValue_1),16) + WORD_TO_UDINT(wInputValue_2);
ELSE
	udiOutputValue := SHL(WORD_TO_UDINT(wInputValue_2),16) + WORD_TO_UDINT(wInputValue_1);
END_IF

END_FUNCTION_BLOCK

// ---- General/FBs Internal/Convert/ULINT/FB_CV_ULINT_TO_WORD.TcPOU
{attribute 'conditionalshow'}
FUNCTION_BLOCK FB_CV_ULINT_TO_WORD
VAR_INPUT
	{attribute 'hide'}
	uliInputValue				: ULINT;							//Input value that is converted into the output value			
	{attribute 'hide'}				
	eByteOrderForConvert		: eByteOrder;						//Byte Format
END_VAR
VAR_OUTPUT
	{attribute 'hide'}
	wOutputValue_1				: WORD;								//Converted output value
	{attribute 'hide'}
	wOutputValue_2				: WORD;								//Converted output value
	{attribute 'hide'}
	wOutputValue_3				: WORD;								//Converted output value
	{attribute 'hide'}
	wOutputValue_4				: WORD;								//Converted output value
END_VAR
VAR
END_VAR

//Creator : Kai Ebensperger
//Company : Lynus AG
//Date : 28.04.2021
//Version : 1.0.0.0

//With this functionblock its possible to convert a certain Datatyp in a other Datatype
//The byte order can be selected between BigEndian and LittleEndian
//ULINT TO WORD
//Created for the Edge Device Lib over Modbus TCP
//Modbus TCP is WORD oriented

IF eByteOrderForConvert = eByteOrder.eBigEndian THEN
	wOutputValue_1 := ULINT_TO_WORD(SHR(uliInputValue,48) AND 16#FFFF);
	wOutputValue_2 := ULINT_TO_WORD(SHR(uliInputValue,32) AND 16#FFFF);
	wOutputValue_3 := ULINT_TO_WORD(SHR(uliInputValue,16) AND 16#FFFF);
	wOutputValue_4 := ULINT_TO_WORD(uliInputValue) AND 16#FFFF;
ELSE
	wOutputValue_4 := ULINT_TO_WORD(SHR(uliInputValue,48) AND 16#FFFF);
	wOutputValue_3 := ULINT_TO_WORD(SHR(uliInputValue,32) AND 16#FFFF);
	wOutputValue_2 := ULINT_TO_WORD(SHR(uliInputValue,16) AND 16#FFFF);
	wOutputValue_1 := ULINT_TO_WORD(uliInputValue) AND 16#FFFF;
END_IF

END_FUNCTION_BLOCK

// ---- General/FBs Internal/Convert/ULINT/FB_CV_WORD_TO_ULINT.TcPOU
{attribute 'conditionalshow'}
FUNCTION_BLOCK FB_CV_WORD_TO_ULINT
VAR_INPUT
	{attribute 'hide'}
	wInputValue_1				: WORD;								//Input value that is converted into the output value
	{attribute 'hide'}
	wInputValue_2				: WORD;								//Input value that is converted into the output value
	{attribute 'hide'}
	wInputValue_3				: WORD;								//Input value that is converted into the output value
	{attribute 'hide'}
	wInputValue_4				: WORD;								//Input value that is converted into the output value
	{attribute 'hide'}
	eByteOrderForConvert		: eByteOrder;						//Byte Format
END_VAR
VAR_OUTPUT
	{attribute 'hide'}
	uliOutputValue				: ULINT;							//Converted output value							
END_VAR
VAR
END_VAR

//Creator : Kai Ebensperger
//Company : Lynus AG
//Date : 28.04.2021
//Version : 1.0.0.0

//With this functionblock its possible to convert a certain Datatyp in a other Datatype
//The byte order can be selected between BigEndian and LittleEndian
//WORD TO ULINT
//Created for the Edge Device Lib over Modbus TCP
//Modbus TCP is WORD oriented

IF eByteOrderForConvert = eByteOrder.eBigEndian THEN
	uliOutputValue := SHL(WORD_TO_ULINT(wInputValue_1),48) + SHL(WORD_TO_ULINT(wInputValue_2),32) + SHL(WORD_TO_ULINT(wInputValue_3),16) + WORD_TO_DWORD(wInputValue_4);
ELSE
	uliOutputValue := SHL(WORD_TO_ULINT(wInputValue_4),48) + SHL(WORD_TO_ULINT(wInputValue_3),32) + SHL(WORD_TO_ULINT(wInputValue_2),16) + WORD_TO_DWORD(wInputValue_1);
END_IF

END_FUNCTION_BLOCK

// ---- General/FBs Internal/Convert/USINT/FB_CV_USINT_TO_WORD.TcPOU
{attribute 'conditionalshow'}
FUNCTION_BLOCK FB_CV_USINT_TO_WORD
VAR_INPUT
	{attribute 'hide'}
	usiInputValue_1				: USINT;								//Input value that is converted into the output value
	{attribute 'hide'}							
	usiInputValue_2				: USINT;								//Input value that is converted into the output value
	{attribute 'hide'}
	eByteOrderForConvert		: eByteOrder;							//Byte Format
END_VAR
VAR_OUTPUT
	{attribute 'hide'}
	wOutputValue				: WORD;									//Converted output value
END_VAR
VAR
END_VAR

//Creator : Kai Ebensperger
//Company : Lynus AG
//Date : 28.04.2021
//Version : 1.0.0.0

//With this functionblock its possible to convert a certain Datatyp in a other Datatype
//The byte order can be selected between BigEndian and LittleEndian
//USINT TO WORD
//Created for the Edge Device Lib over Modbus TCP
//Modbus TCP is WORD oriented

IF eByteOrderForConvert = eByteOrder.eBigEndian THEN
	wOutputValue := SHL(USINT_TO_WORD(usiInputValue_1),8) + USINT_TO_WORD(usiInputValue_2);
ELSE
	wOutputValue := SHL(USINT_TO_WORD(usiInputValue_2),8) + USINT_TO_WORD(usiInputValue_1);
END_IF

END_FUNCTION_BLOCK

// ---- General/FBs Internal/Convert/USINT/FB_CV_WORD_TO_USINT.TcPOU
{attribute 'conditionalshow'}
FUNCTION_BLOCK FB_CV_WORD_TO_USINT
VAR_INPUT
	{attribute 'hide'}
	wInputValue					: WORD;									//Input value that is converted into the output value
	{attribute 'hide'}
	eByteOrderForConvert		: eByteOrder;							//Byte Format
END_VAR
VAR_OUTPUT
	{attribute 'hide'}
	usiOutputValue_1			: USINT;								//Converted output value	
	{attribute 'hide'}						
	usiOutputValue_2			: USINT;								//Converted output value
END_VAR
VAR
END_VAR

//Creator : Kai Ebensperger
//Company : Lynus AG
//Date : 28.04.2021
//Version : 1.0.0.0

//With this functionblock its possible to convert a certain Datatyp in a other Datatype
//The byte order can be selected between BigEndian and LittleEndian
//WORD TO USINT
//Created for the Edge Device Lib over Modbus TCP
//Modbus TCP is WORD oriented

IF eByteOrderForConvert = eByteOrder.eBigEndian THEN
	usiOutputValue_1 := WORD_TO_USINT(SHR(wInputValue,8) AND 16#FFFF);
	usiOutputValue_2 := WORD_TO_USINT(wInputValue AND 16#FFFF);
ELSE
	usiOutputValue_2 := WORD_TO_USINT(SHR(wInputValue,8) AND 16#FFFF);
	usiOutputValue_1 := WORD_TO_USINT(wInputValue AND 16#FFFF);
END_IF

END_FUNCTION_BLOCK

// ---- General/FBs Internal/Filter/FB_Filter.TcPOU
{attribute 'hide_all_locals'}
{attribute 'conditionalshow'}
FUNCTION_BLOCK FB_Filter
//Arithmetic moving average 			 (Simple Moving Average, SMA)
VAR_INPUT
	{attribute 'hide'}
	x		: REAL;						//Value to be filtered and annealed
	{attribute 'hide'}
	tm		: INT := 100; 				//messurement delay [ms]
	{attribute 'hide'}
	k		: INT := 10; 				//maximal count of values max 1000
	{attribute 'hide'}
	tbase 	: TIME := T#1MS; 			//Time delay between values
END_VAR
VAR CONSTANT
	{attribute 'hide'}
	LIM 	: INT := 1000; 				//Limit of values = 1000
END_VAR
VAR_OUTPUT
	{attribute 'hide'}
	y		: REAL;						//Filtered and smoothed value
END_VAR
VAR
	DELAY 	: TON;						//Timer for time delay
	values 	: ARRAY [0..1000] OF REAL;	//Array with the values
	i  		: INT;						//Auxiliary variable for array
END_VAR

//Filter that writes a certain number of values to an array over a configurable time.
delay(IN := TRUE,PT:= tbase * tm );

k := LIMIT(0,k,1000);
	k := MAX(k,1);

IF DELAY.Q THEN

	delay(IN:=FALSE);

	k := MIN(k,LIM);

	values[i] :=x;
		i := i + 1;
			IF i > k THEN i := 0; END_IF;
END_IF

y := ARRAY_AVG(ADR(values), INT_TO_UINT(K*4));

END_FUNCTION_BLOCK

// ---- General/FUNs Internal/ARRAY_AVG.TcPOU
{attribute 'conditionalshow'}
FUNCTION ARRAY_AVG : REAL
VAR_INPUT
	{attribute 'hide'}
	pt   	: POINTER TO ARRAY[0..32000] OF REAL;			//Pointer with the content
	{attribute 'hide'}
	size 	: UINT;											//Size of the data
END_VAR
VAR
	{attribute 'hide'}
	i		: UINT;											//loop internal
	{attribute 'hide'}
	stop	: UINT;											//End of the loop
END_VAR

//this function will calculate the average of a given array.
//the function needs to be called:	array_avg(adr("array"),sizeof("array"));
//because this function works with pointers its very time efficient and it needs no extra memory.

//ARRAY AVG function calculates the mean value of an arbitrary real array
stop := SHR(size,2)-1;
	IF stop = 0 THEN
		ARRAY_AVG := (pt^[0] + pt^[1]) / 2;
	ELSE
		ARRAY_AVG := pt^[0];
	END_IF
		IF stop > 0 AND stop <= 32000 THEN		
			FOR i := 1 TO stop DO
				ARRAY_AVG := ARRAY_AVG + pt^[i];
			END_FOR;
		END_IF
			ARRAY_AVG := ARRAY_AVG / UINT_TO_REAL(stop + 1);

END_FUNCTION

// ---- General/FBs Internal/Linear Interpolation/FB_Lin_Interpolation.TcPOU
{attribute 'hide_all_locals'}
{attribute 'conditionalshow'}
FUNCTION_BLOCK FB_Lin_Interpolation
VAR_INPUT
	{attribute 'hide'}
	rXInputValue				: REAL;													//X Input Value from which the Y value is to be determined 
	{attribute 'hide'}
	arrXIntermediateValues		: ARRAY[1..10] OF REAL;									//X Intermediate Values
	{attribute 'hide'}
	arrYIntermediateValues		: ARRAY[1..10] OF REAL;									//Y Intermediate Values
END_VAR
VAR_OUTPUT
	{attribute 'hide'}
	rYOutputValue				: REAL;													//Y Output Value
END_VAR
VAR
	rY1							: REAL;													//Internal value for calculation
	rY2							: REAL;													//Internal value for calculation
	rX1							: REAL;													//Internal value for calculation
	rX2							: REAL;													//Internal value for calculation
END_VAR

//Creator : Kai Ebensperger
//Company : Lynus AG
//Date : 04.10.2021
//Version : 1.0.0.0

//With this function it is possible to change a linear value to a non-linear output value using linear interpolation.
//The X value and the X Array are the are know
//The Y array refers to the value you want to have as output value and always refers in position to the X array. So XArray[1] = YArray[1] etc...
//All values in between are calculated

IF rXInputValue >= 0 AND rXInputValue <= arrXIntermediateValues[1] THEN
	rX1 := 0; rX2 :=  arrXIntermediateValues[1];
		rY1 := 0; rY2 := arrYIntermediateValues[1];
ELSIF rXInputValue > arrXIntermediateValues[1] AND rXInputValue <= arrXIntermediateValues[2] THEN
	rX1 :=  arrXIntermediateValues[1]; rX2 := arrXIntermediateValues[2];
		rY1 := arrYIntermediateValues[1]; rY2 := arrYIntermediateValues[2];
ELSIF rXInputValue > arrXIntermediateValues[2] AND rXInputValue <= arrXIntermediateValues[3] THEN
	rX1 :=  arrXIntermediateValues[2]; rX2 := arrXIntermediateValues[3];
		rY1 := arrYIntermediateValues[2]; rY2 := arrYIntermediateValues[3];
ELSIF rXInputValue > arrXIntermediateValues[3] AND rXInputValue <= arrXIntermediateValues[4] THEN
	rX1 :=  arrXIntermediateValues[3]; rX2 := arrXIntermediateValues[4];
		rY1 := arrYIntermediateValues[3]; rY2 := arrYIntermediateValues[4];
ELSIF rXInputValue > arrXIntermediateValues[4] AND rXInputValue <= arrXIntermediateValues[5] THEN
	rX1 :=  arrXIntermediateValues[4]; rX2 := arrXIntermediateValues[5];
		rY1 := arrYIntermediateValues[4]; rY2 := arrYIntermediateValues[5];
ELSIF rXInputValue > arrXIntermediateValues[5] AND rXInputValue <= arrXIntermediateValues[6] THEN
	rX1 :=  arrXIntermediateValues[5]; rX2 := arrXIntermediateValues[6];
		rY1 := arrYIntermediateValues[5]; rY2 := arrYIntermediateValues[6];
ELSIF rXInputValue > arrXIntermediateValues[6] AND rXInputValue <= arrXIntermediateValues[7] THEN
	rX1 :=  arrXIntermediateValues[6]; rX2 := arrXIntermediateValues[7];
		rY1 := arrYIntermediateValues[6]; rY2 := arrYIntermediateValues[7];
ELSIF rXInputValue > arrXIntermediateValues[7] AND rXInputValue <= arrXIntermediateValues[8] THEN
	rX1 :=  arrXIntermediateValues[7]; rX2 := arrXIntermediateValues[8];
		rY1 := arrYIntermediateValues[7]; rY2 := arrYIntermediateValues[8];
ELSIF rXInputValue > arrXIntermediateValues[8] AND rXInputValue <= arrXIntermediateValues[9] THEN
	rX1 :=  arrXIntermediateValues[8]; rX2 := arrXIntermediateValues[9];
		rY1 := arrYIntermediateValues[8]; rY2 := arrYIntermediateValues[9];
ELSIF rXInputValue > arrXIntermediateValues[9] AND rXInputValue <= arrXIntermediateValues[10] THEN
	rX1 :=  arrXIntermediateValues[9]; rX2 := arrXIntermediateValues[10];
		rY1 := arrYIntermediateValues[9]; rY2 := arrYIntermediateValues[10];
END_IF

rYOutputValue := F_Scalvalue(x:= rXInputValue, x1:= rX1, y1:= rY1, x2:= rX2, y2:= rY2);
	rYOutputValue := LIMIT(rY1,rYOutputValue,rY2);

END_FUNCTION_BLOCK

// ---- General/FBs Internal/Number Of Device/FB_NumberOfDevice.TcPOU
{attribute 'hide_all_locals'}
{attribute 'conditionalshow'}
FUNCTION_BLOCK FB_NumberOfDevice
VAR_INPUT
	{attribute 'hide'}
	diActualNumberOfDevices			: DINT;							//Actual Number for this Device
	{attribute 'hide'}
	diMaxNumberOfDevices			: DINT;							//Max Numbers for this Device
	{attribute 'hide'}
	udiCounterOnlineChange			: UDINT;						//Actual Counter for Online change
END_VAR
VAR_OUTPUT
	{attribute 'hide'}
	bNumberIsCalculatet				: BOOL;							//Number for this Device ic calculatet
	{attribute 'hide'}
	bFPNumberIsCalculatet			: BOOL;							//Number for this Device ic calculatet. Only positive Edge
	{attribute 'hide'}
	bOnlineChange					: BOOL;							//Its true for 1 cycle when a Online change was success
	{attribute 'hide'}
	diNumberForThisDevice			: DINT;							//Number for this Device
	{attribute 'hide'}
	diNumberOfTotalDevices			: DINT;							//Total Devices without Limits
END_VAR
VAR
	FPCalculatet					: R_TRIG;						//Internal positive edge
	udiCounterOnlineChange_CP		: UDINT;						//Counter online changen to compare with the original input variable
END_VAR

//Creator : Kai Ebensperger
//Company : Lynus AG
//Date : 29.05.2021
//Version : 1.0.0.0

//With this Function its possible to count a number for a Device in PLC
//The number reset and renew when we have a online change on the plc

